LIN {X 0,Y 287.469,Z 770.66,A -85,B 0,C 180,E1 15282.197,E2 15282.197} C_VEL
LIN {X 0,Y 284.222,Z 794.755,A -85,B 0,C 180,E1 15292.332,E2 15292.332} C_VEL
LIN {X 0,Y 283.558,Z 803.475,A -85,B 0,C 180,E1 15301.536,E2 15301.536} C_VEL
LIN {X 0,Y 286.517,Z 800.266,A -85,B 0,C 180,E1 15312.078,E2 15312.078} C_VEL
LIN {X 0,Y 295.291,Z 782.461,A -85,B 0,C 180,E1 15322.672,E2 15322.672} C_VEL
LIN {X 0,Y 310.882,Z 750.712,A -85,B 0,C 180,E1 15331.653,E2 15331.653} C_VEL
LIN {X 0,Y 330.925,Z 705.593,A -85,B 0,C 180,E1 15338.602,E2 15338.602} C_VEL
LIN {X 0,Y 336.814,Z 689.201,A -85,B 0,C 180,E1 15340.792,E2 15340.792} C_VEL
LIN {X 0,Y 337.476,Z 683.839,A -85,B 0,C 180,E1 15344.187,E2 15344.187} C_VEL
LIN {X 0,Y 338.249,Z 688.288,A -85,B 0,C 180,E1 15347.754,E2 15347.754} C_VEL
LIN {X 0,Y 313.848,Z 750.158,A -85,B 0,C 180,E1 15354.353,E2 15354.353} C_VEL
LIN {X 0,Y 295.88,Z 793.344,A -85,B 0,C 180,E1 15362.953,E2 15362.953} C_VEL
LIN {X 0,Y 286.115,Z 820.837,A -85,B 0,C 180,E1 15373.067,E2 15373.067} C_VEL
LIN {X 0,Y 283.836,Z 832.792,A -85,B 0,C 180,E1 15382.345,E2 15382.345} C_VEL
LIN {X 0,Y 283.962,Z 833.571,A -85,B 0,C 180,E1 15391.556,E2 15391.556} C_VEL
LIN {X 0,Y 284.286,Z 822.206,A -85,B 0,C 180,E1 15400.792,E2 15400.792} C_VEL
LIN {X 0,Y 287.24,Z 796.191,A -85,B 0,C 180,E1 15410.108,E2 15410.108} C_VEL
LIN {X 0,Y 300.181,Z 753.134,A -85,B 0,C 180,E1 15421.206,E2 15421.206} C_VEL
LIN {X 0,Y 316.341,Z 705.619,A -85,B 0,C 180,E1 15427.781,E2 15427.781} C_VEL
LIN {X 0,Y 323.777,Z 675.076,A -85,B 0,C 180,E1 15430.595,E2 15430.595} C_VEL
LIN {X 0,Y 318.954,Z 657.733,A -85,B 0,C 180,E1 15435.308,E2 15435.308} C_VEL
LIN {X 0,Y 315.945,Z 652.697,A -85,B 0,C 180,E1 15439.832,E2 15439.832} C_VEL
LIN {X 0,Y 312.951,Z 664.798,A -85,B 0,C 180,E1 15445.963,E2 15445.963} C_VEL
LIN {X 0,Y 312.289,Z 682.68,A -85,B 0,C 180,E1 15451.384,E2 15451.384} C_VEL
LIN {X 0,Y 297.451,Z 717.791,A -85,B 0,C 180,E1 15458.29,E2 15458.29} C_VEL
LIN {X 0,Y 286.13,Z 736.914,A -85,B 0,C 180,E1 15466.19,E2 15466.19} C_VEL
LIN {X 0,Y 279.764,Z 741.327,A -85,B 0,C 180,E1 15475.331,E2 15475.331} C_VEL
LIN {X 0,Y 278.19,Z 731.042,A -85,B 0,C 180,E1 15483.907,E2 15483.907} C_VEL
LIN {X 0,Y 279.775,Z 705.474,A -85,B 0,C 180,E1 15492.228,E2 15492.228} C_VEL
LIN {X 0,Y 283.473,Z 665.617,A -85,B 0,C 180,E1 15498.935,E2 15498.935} C_VEL
LIN {X 0,Y 281.601,Z 639.243,A -85,B 0,C 180,E1 15501.747,E2 15501.747} C_VEL
LIN {X 0,Y 273.533,Z 602.81,A -85,B 0,C 180,E1 15504.584,E2 15504.584} C_VEL
LIN {X 0,Y 272.564,Z 602.81,A -85,B 0,C 180,E1 15516.131,E2 15516.131} C_VEL
LIN {X 0,Y 272.447,Z 602.81,A -85,B 0,C 180,E1 15530.139,E2 15530.139} C_VEL
LIN {X 0,Y 272.833,Z 602.81,A -85,B 0,C 180,E1 15541.759,E2 15541.759} C_VEL
LIN {X 0,Y 273.836,Z 602.81,A -85,B 0,C 180,E1 15555.866,E2 15555.866} C_VEL
LIN {X 0,Y 275.222,Z 602.81,A -85,B 0,C 180,E1 15568.395,E2 15568.395} C_VEL
LIN {X 0,Y 274.237,Z 602.81,A -85,B 0,C 180,E1 15581.14,E2 15581.14} C_VEL
LIN {X 0,Y 273.286,Z 602.81,A -85,B 0,C 180,E1 15594.58,E2 15594.58} C_VEL
LIN {X 0,Y 272.71,Z 602.81,A -85,B 0,C 180,E1 15606.216,E2 15606.216} C_VEL
LIN {X 0,Y 272.978,Z 604.085,A -85,B 0,C 180,E1 15619.483,E2 15619.483} C_VEL
LIN {X 0,Y 292.995,Z 665.219,A -85,B 0,C 180,E1 15624.943,E2 15624.943} C_VEL
LIN {X 0,Y 295.039,Z 684.173,A -85,B 0,C 180,E1 15626.919,E2 15626.919} C_VEL
LIN {X 0,Y 286.379,Z 734.413,A -85,B 0,C 180,E1 15633.535,E2 15633.535} C_VEL
LIN {X 0,Y 279.424,Z 771.619,A -85,B 0,C 180,E1 15642.226,E2 15642.226} C_VEL
LIN {X 0,Y 276.273,Z 794.637,A -85,B 0,C 180,E1 15652.11,E2 15652.11} C_VEL
LIN {X 0,Y 275.575,Z 803.87,A -85,B 0,C 180,E1 15661.58,E2 15661.58} C_VEL
LIN {X 0,Y 278.805,Z 801.152,A -85,B 0,C 180,E1 15672.577,E2 15672.577} C_VEL
LIN {X 0,Y 288.146,Z 784.349,A -85,B 0,C 180,E1 15683.267,E2 15683.267} C_VEL
LIN {X 0,Y 305.45,Z 752.594,A -85,B 0,C 180,E1 15692.705,E2 15692.705} C_VEL
LIN {X 0,Y 327.249,Z 708.48,A -85,B 0,C 180,E1 15699.733,E2 15699.733} C_VEL
LIN {X 0,Y 332.934,Z 695.38,A -85,B 0,C 180,E1 15701.371,E2 15701.371} C_VEL
LIN {X 0,Y 334.073,Z 691.222,A -85,B 0,C 180,E1 15704.757,E2 15704.757} C_VEL
LIN {X 0,Y 334.163,Z 694.797,A -85,B 0,C 180,E1 15707.115,E2 15707.115} C_VEL
LIN {X 0,Y 309.62,Z 749.376,A -85,B 0,C 180,E1 15712.915,E2 15712.915} C_VEL
LIN {X 0,Y 289.453,Z 793.221,A -85,B 0,C 180,E1 15721.877,E2 15721.877} C_VEL
LIN {X 0,Y 278.386,Z 821.027,A -85,B 0,C 180,E1 15732.582,E2 15732.582} C_VEL
LIN {X 0,Y 275.855,Z 832.48,A -85,B 0,C 180,E1 15742.122,E2 15742.122} C_VEL
LIN {X 0,Y 275.993,Z 832.853,A -85,B 0,C 180,E1 15751.601,E2 15751.601} C_VEL
LIN {X 0,Y 276.307,Z 820.985,A -85,B 0,C 180,E1 15761.108,E2 15761.108} C_VEL
LIN {X 0,Y 279.561,Z 794.339,A -85,B 0,C 180,E1 15770.686,E2 15770.686} C_VEL
LIN {X 0,Y 292.103,Z 757.137,A -85,B 0,C 180,E1 15781.346,E2 15781.346} C_VEL
LIN {X 0,Y 309.645,Z 710.546,A -85,B 0,C 180,E1 15788.433,E2 15788.433} C_VEL
LIN {X 0,Y 318.887,Z 677.805,A -85,B 0,C 180,E1 15791.672,E2 15791.672} C_VEL
LIN {X 0,Y 314.799,Z 662.667,A -85,B 0,C 180,E1 15796.655,E2 15796.655} C_VEL
LIN {X 0,Y 312.531,Z 660.915,A -85,B 0,C 180,E1 15803.272,E2 15803.272} C_VEL
LIN {X 0,Y 312.951,Z 664.798,A -85,B 0,C 180,E1 15805.963,E2 15805.963} C_VEL
LIN {X 0,Y 308.353,Z 681.058,A -85,B 0,C 180,E1 15809.107,E2 15809.107} C_VEL
LIN {X 0,Y 300.727,Z 701.492,A -85,B 0,C 180,E1 15812.988,E2 15812.988} C_VEL
LIN {X 0,Y 285.864,Z 729.53,A -85,B 0,C 180,E1 15820.621,E2 15820.621} C_VEL
LIN {X 0,Y 275.928,Z 742.078,A -85,B 0,C 180,E1 15828.9,E2 15828.9} C_VEL
LIN {X 0,Y 271.169,Z 740.21,A -85,B 0,C 180,E1 15838.394,E2 15838.394} C_VEL
LIN {X 0,Y 270.306,Z 723.721,A -85,B 0,C 180,E1 15847.254,E2 15847.254} C_VEL
LIN {X 0,Y 272.947,Z 691.929,A -85,B 0,C 180,E1 15855.31,E2 15855.31} C_VEL
LIN {X 0,Y 275.844,Z 650.722,A -85,B 0,C 180,E1 15860.949,E2 15860.949} C_VEL
LIN {X 0,Y 265.38,Z 602.81,A -85,B 0,C 180,E1 15865.13,E2 15865.13} C_VEL
LIN {X 0,Y 264.414,Z 602.81,A -85,B 0,C 180,E1 15879.179,E2 15879.179} C_VEL
LIN {X 0,Y 264.42,Z 602.81,A -85,B 0,C 180,E1 15892.915,E2 15892.915} C_VEL
LIN {X 0,Y 264.872,Z 602.81,A -85,B 0,C 180,E1 15904.525,E2 15904.525} C_VEL
LIN {X 0,Y 266.041,Z 602.81,A -85,B 0,C 180,E1 15918.458,E2 15918.458} C_VEL
LIN {X 0,Y 266.94,Z 602.81,A -85,B 0,C 180,E1 15931.602,E2 15931.602} C_VEL
LIN {X 0,Y 265.894,Z 602.81,A -85,B 0,C 180,E1 15944.853,E2 15944.853} C_VEL
LIN {X 0,Y 265.023,Z 602.81,A -85,B 0,C 180,E1 15957.445,E2 15957.445} C_VEL
LIN {X 0,Y 264.599,Z 602.81,A -85,B 0,C 180,E1 15971.224,E2 15971.224} C_VEL
LIN {X 0,Y 264.888,Z 603.872,A -85,B 0,C 180,E1 15978.645,E2 15978.645} C_VEL
LIN {X 0,Y 284.837,Z 664.739,A -85,B 0,C 180,E1 15984.251,E2 15984.251} C_VEL
LIN {X 0,Y 287.376,Z 685.203,A -85,B 0,C 180,E1 15986.469,E2 15986.469} C_VEL
LIN {X 0,Y 278.443,Z 735.564,A -85,B 0,C 180,E1 15993.321,E2 15993.321} C_VEL
LIN {X 0,Y 271.266,Z 773.261,A -85,B 0,C 180,E1 16002.504,E2 16002.504} C_VEL
LIN {X 0,Y 268.205,Z 795.774,A -85,B 0,C 180,E1 16012.689,E2 16012.689} C_VEL
LIN {X 0,Y 267.587,Z 804.24,A -85,B 0,C 180,E1 16021.627,E2 16021.627} C_VEL
LIN {X 0,Y 271.036,Z 802.205,A -85,B 0,C 180,E1 16032.944,E2 16032.944} C_VEL
LIN {X 0,Y 282.031,Z 784.649,A -85,B 0,C 180,E1 16044.647,E2 16044.647} C_VEL
LIN {X 0,Y 301.744,Z 752.031,A -85,B 0,C 180,E1 16054.371,E2 16054.371} C_VEL
LIN {X 0,Y 326.723,Z 706.2,A -85,B 0,C 180,E1 16061.502,E2 16061.502} C_VEL
LIN {X 0,Y 329.631,Z 699.986,A -85,B 0,C 180,E1 16062.496,E2 16062.496} C_VEL
LIN {X 0,Y 330.683,Z 699.253,A -85,B 0,C 180,E1 16066.028,E2 16066.028} C_VEL
LIN {X 0,Y 304.263,Z 751.972,A -85,B 0,C 180,E1 16071.922,E2 16071.922} C_VEL
LIN {X 0,Y 282.512,Z 794.499,A -85,B 0,C 180,E1 16081.122,E2 16081.122} C_VEL
LIN {X 0,Y 270.691,Z 821.198,A -85,B 0,C 180,E1 16092.071,E2 16092.071} C_VEL
LIN {X 0,Y 267.82,Z 832.451,A -85,B 0,C 180,E1 16102.568,E2 16102.568} C_VEL
LIN {X 0,Y 268.044,Z 832.084,A -85,B 0,C 180,E1 16111.648,E2 16111.648} C_VEL
LIN {X 0,Y 268.378,Z 819.679,A -85,B 0,C 180,E1 16121.44,E2 16121.44} C_VEL
LIN {X 0,Y 281.539,Z 767.173,A -85,B 0,C 180,E1 16139.932,E2 16139.932} C_VEL
LIN {X 0,Y 298.719,Z 725.735,A -85,B 0,C 180,E1 16147.805,E2 16147.805} C_VEL
LIN {X 0,Y 314.035,Z 681.623,A -85,B 0,C 180,E1 16152.674,E2 16152.674} C_VEL
LIN {X 0,Y 310.873,Z 668.739,A -85,B 0,C 180,E1 16157.638,E2 16157.638} C_VEL
LIN {X 0,Y 309.011,Z 669.222,A -85,B 0,C 180,E1 16164.156,E2 16164.156} C_VEL
LIN {X 0,Y 308.353,Z 681.058,A -85,B 0,C 180,E1 16169.107,E2 16169.107} C_VEL
LIN {X 0,Y 297.981,Z 699.899,A -85,B 0,C 180,E1 16171.12,E2 16171.12} C_VEL
LIN {X 0,Y 281.339,Z 728.984,A -85,B 0,C 180,E1 16178.647,E2 16178.647} C_VEL
LIN {X 0,Y 269.649,Z 742.928,A -85,B 0,C 180,E1 16186.988,E2 16186.988} C_VEL
LIN {X 0,Y 263.562,Z 742.734,A -85,B 0,C 180,E1 16196.697,E2 16196.697} C_VEL
LIN {X 0,Y 262.364,Z 727.153,A -85,B 0,C 180,E1 16206.223,E2 16206.223} C_VEL
LIN {X 0,Y 264.607,Z 696.697,A -85,B 0,C 180,E1 16214.649,E2 16214.649} C_VEL
LIN {X 0,Y 268.302,Z 653.679,A -85,B 0,C 180,E1 16220.996,E2 16220.996} C_VEL
LIN {X 0,Y 257.235,Z 602.81,A -85,B 0,C 180,E1 16225.746,E2 16225.746} C_VEL
LIN {X 0,Y 256.407,Z 602.81,A -85,B 0,C 180,E1 16238.416,E2 16238.416} C_VEL
LIN {X 0,Y 256.424,Z 602.81,A -85,B 0,C 180,E1 16253.022,E2 16253.022} C_VEL
LIN {X 0,Y 256.979,Z 602.81,A -85,B 0,C 180,E1 16267.401,E2 16267.401} C_VEL
LIN {X 0,Y 258.297,Z 602.81,A -85,B 0,C 180,E1 16281.527,E2 16281.527} C_VEL
LIN {X 0,Y 258.955,Z 602.81,A -85,B 0,C 180,E1 16291.651,E2 16291.651} C_VEL
LIN {X 0,Y 257.807,Z 602.81,A -85,B 0,C 180,E1 16305.33,E2 16305.33} C_VEL
LIN {X 0,Y 257.047,Z 602.81,A -85,B 0,C 180,E1 16316.247,E2 16316.247} C_VEL
LIN {X 0,Y 256.544,Z 602.81,A -85,B 0,C 180,E1 16328.356,E2 16328.356} C_VEL
LIN {X 0,Y 256.908,Z 604.687,A -85,B 0,C 180,E1 16337.833,E2 16337.833} C_VEL
LIN {X 0,Y 276.651,Z 664.319,A -85,B 0,C 180,E1 16343.539,E2 16343.539} C_VEL
LIN {X 0,Y 279.656,Z 686.55,A -85,B 0,C 180,E1 16346.047,E2 16346.047} C_VEL
LIN {X 0,Y 270.659,Z 735.793,A -85,B 0,C 180,E1 16352.94,E2 16352.94} C_VEL
LIN {X 0,Y 263.268,Z 773.811,A -85,B 0,C 180,E1 16362.454,E2 16362.454} C_VEL
LIN {X 0,Y 260.096,Z 796.908,A -85,B 0,C 180,E1 16373.361,E2 16373.361} C_VEL
LIN {X 0,Y 259.598,Z 804.598,A -85,B 0,C 180,E1 16381.677,E2 16381.677} C_VEL
LIN {X 0,Y 263.289,Z 803.29,A -85,B 0,C 180,E1 16393.332,E2 16393.332} C_VEL
LIN {X 0,Y 275.056,Z 786.755,A -85,B 0,C 180,E1 16405.316,E2 16405.316} C_VEL
LIN {X 0,Y 296.941,Z 754.215,A -85,B 0,C 180,E1 16415.545,E2 16415.545} C_VEL
LIN {X 0,Y 324.272,Z 709.128,A -85,B 0,C 180,E1 16422.733,E2 16422.733} C_VEL
LIN {X 0,Y 326.195,Z 705.607,A -85,B 0,C 180,E1 16423.893,E2 16423.893} C_VEL
LIN {X 0,Y 325.813,Z 706.997,A -85,B 0,C 180,E1 16425.196,E2 16425.196} C_VEL
LIN {X 0,Y 298.501,Z 755.637,A -85,B 0,C 180,E1 16431.05,E2 16431.05} C_VEL
LIN {X 0,Y 274.994,Z 797.097,A -85,B 0,C 180,E1 16440.708,E2 16440.708} C_VEL
LIN {X 0,Y 262.288,Z 823.151,A -85,B 0,C 180,E1 16452.68,E2 16452.68} C_VEL
LIN {X 0,Y 259.893,Z 831.729,A -85,B 0,C 180,E1 16461.635,E2 16461.635} C_VEL
LIN {X 0,Y 260.078,Z 831.237,A -85,B 0,C 180,E1 16471.699,E2 16471.699} C_VEL
LIN {X 0,Y 260.423,Z 818.323,A -85,B 0,C 180,E1 16481.795,E2 16481.795} C_VEL
LIN {X 0,Y 275.82,Z 764.726,A -85,B 0,C 180,E1 16501.538,E2 16501.538} C_VEL
LIN {X 0,Y 295.082,Z 722.453,A -85,B 0,C 180,E1 16509.512,E2 16509.512} C_VEL
LIN {X 0,Y 309.243,Z 685.758,A -85,B 0,C 180,E1 16513.651,E2 16513.651} C_VEL
LIN {X 0,Y 307.017,Z 675.555,A -85,B 0,C 180,E1 16518.141,E2 16518.141} C_VEL
LIN {X 0,Y 304.98,Z 677.854,A -85,B 0,C 180,E1 16525.094,E2 16525.094} C_VEL
LIN {X 0,Y 301.801,Z 692.035,A -85,B 0,C 180,E1 16529.805,E2 16529.805} C_VEL
LIN {X 0,Y 297.981,Z 699.899,A -85,B 0,C 180,E1 16531.12,E2 16531.12} C_VEL
LIN {X 0,Y 284.761,Z 717.187,A -85,B 0,C 180,E1 16533.109,E2 16533.109} C_VEL
LIN {X 0,Y 268.1,Z 739.787,A -85,B 0,C 180,E1 16541.859,E2 16541.859} C_VEL
LIN {X 0,Y 258.235,Z 746.307,A -85,B 0,C 180,E1 16551.55,E2 16551.55} C_VEL
LIN {X 0,Y 254.341,Z 738.641,A -85,B 0,C 180,E1 16560.852,E2 16560.852} C_VEL
LIN {X 0,Y 254.813,Z 716.975,A -85,B 0,C 180,E1 16569.941,E2 16569.941} C_VEL
LIN {X 0,Y 258.316,Z 681.012,A -85,B 0,C 180,E1 16577.74,E2 16577.74} C_VEL
LIN {X 0,Y 259.305,Z 648.919,A -85,B 0,C 180,E1 16581.909,E2 16581.909} C_VEL
LIN {X 0,Y 249.167,Z 602.81,A -85,B 0,C 180,E1 16586.093,E2 16586.093} C_VEL
LIN {X 0,Y 248.259,Z 602.81,A -85,B 0,C 180,E1 16600.138,E2 16600.138} C_VEL
LIN {X 0,Y 248.454,Z 602.81,A -85,B 0,C 180,E1 16615.536,E2 16615.536} C_VEL
LIN {X 0,Y 249.223,Z 602.81,A -85,B 0,C 180,E1 16630.686,E2 16630.686} C_VEL
LIN {X 0,Y 250.622,Z 602.81,A -85,B 0,C 180,E1 16644.761,E2 16644.761} C_VEL
LIN {X 0,Y 250.703,Z 602.81,A -85,B 0,C 180,E1 16655.18,E2 16655.18} C_VEL
LIN {X 0,Y 249.457,Z 602.81,A -85,B 0,C 180,E1 16669.515,E2 16669.515} C_VEL
LIN {X 0,Y 248.59,Z 602.81,A -85,B 0,C 180,E1 16684.509,E2 16684.509} C_VEL
LIN {X 0,Y 248.68,Z 604.118,A -85,B 0,C 180,E1 16696.888,E2 16696.888} C_VEL
LIN {X 0,Y 268.789,Z 665.113,A -85,B 0,C 180,E1 16702.941,E2 16702.941} C_VEL
LIN {X 0,Y 271.898,Z 688.181,A -85,B 0,C 180,E1 16705.647,E2 16705.647} C_VEL
LIN {X 0,Y 262.515,Z 737.945,A -85,B 0,C 180,E1 16712.926,E2 16712.926} C_VEL
LIN {X 0,Y 255.286,Z 774.347,A -85,B 0,C 180,E1 16722.417,E2 16722.417} C_VEL
LIN {X 0,Y 252.05,Z 797.428,A -85,B 0,C 180,E1 16733.644,E2 16733.644} C_VEL
LIN {X 0,Y 252.274,Z 806.144,A -85,B 0,C 180,E1 16745.179,E2 16745.179} C_VEL
LIN {X 0,Y 257.768,Z 801.717,A -85,B 0,C 180,E1 16757.121,E2 16757.121} C_VEL
LIN {X 0,Y 273.27,Z 782.144,A -85,B 0,C 180,E1 16769.074,E2 16769.074} C_VEL
LIN {X 0,Y 300.349,Z 745.184,A -85,B 0,C 180,E1 16779.167,E2 16779.167} C_VEL
LIN {X 0,Y 321.944,Z 712.844,A -85,B 0,C 180,E1 16784.193,E2 16784.193} C_VEL
LIN {X 0,Y 291.755,Z 761.023,A -85,B 0,C 180,E1 16790.456,E2 16790.456} C_VEL
LIN {X 0,Y 266.81,Z 800.691,A -85,B 0,C 180,E1 16800.657,E2 16800.657} C_VEL
LIN {X 0,Y 253.97,Z 824.758,A -85,B 0,C 180,E1 16813.267,E2 16813.267} C_VEL
LIN {X 0,Y 251.82,Z 832.288,A -85,B 0,C 180,E1 16824.843,E2 16824.843} C_VEL
LIN {X 0,Y 252.078,Z 827.384,A -85,B 0,C 180,E1 16835.209,E2 16835.209} C_VEL
LIN {X 0,Y 253.512,Z 808.014,A -85,B 0,C 180,E1 16846.165,E2 16846.165} C_VEL
LIN {X 0,Y 269.716,Z 763.882,A -85,B 0,C 180,E1 16862.816,E2 16862.816} C_VEL
LIN {X 0,Y 290.947,Z 721.586,A -85,B 0,C 180,E1 16870.964,E2 16870.964} C_VEL
LIN {X 0,Y 304.515,Z 690.471,A -85,B 0,C 180,E1 16874.523,E2 16874.523} C_VEL
LIN {X 0,Y 303.557,Z 683.416,A -85,B 0,C 180,E1 16877.553,E2 16877.553} C_VEL
LIN {X 0,Y 301.242,Z 682.497,A -85,B 0,C 180,E1 16882.997,E2 16882.997} C_VEL
LIN {X 0,Y 298.273,Z 693.389,A -85,B 0,C 180,E1 16888.242,E2 16888.242} C_VEL
LIN {X 0,Y 284.761,Z 717.187,A -85,B 0,C 180,E1 16893.109,E2 16893.109} C_VEL
LIN {X 0,Y 266.731,Z 736.601,A -85,B 0,C 180,E1 16897.983,E2 16897.983} C_VEL
LIN {X 0,Y 256.462,Z 745.944,A -85,B 0,C 180,E1 16904.555,E2 16904.555} C_VEL
LIN {X 0,Y 248.297,Z 746.231,A -85,B 0,C 180,E1 16914.737,E2 16914.737} C_VEL
LIN {X 0,Y 246.346,Z 732.566,A -85,B 0,C 180,E1 16924.413,E2 16924.413} C_VEL
LIN {X 0,Y 248.209,Z 703.423,A -85,B 0,C 180,E1 16933.701,E2 16933.701} C_VEL
LIN {X 0,Y 252.493,Z 661.404,A -85,B 0,C 180,E1 16940.801,E2 16940.801} C_VEL
LIN {X 0,Y 243.644,Z 613.537,A -85,B 0,C 180,E1 16945.595,E2 16945.595} C_VEL
LIN {X 0,Y 241.048,Z 602.81,A -85,B 0,C 180,E1 16946.573,E2 16946.573} C_VEL
LIN {X 0,Y 240.089,Z 602.81,A -85,B 0,C 180,E1 16961.575,E2 16961.575} C_VEL
LIN {X 0,Y 240.183,Z 602.81,A -85,B 0,C 180,E1 16973.081,E2 16973.081} C_VEL
LIN {X 0,Y 240.787,Z 602.81,A -85,B 0,C 180,E1 16986.031,E2 16986.031} C_VEL
LIN {X 0,Y 242.16,Z 602.81,A -85,B 0,C 180,E1 17000.958,E2 17000.958} C_VEL
LIN {X 0,Y 242.937,Z 602.81,A -85,B 0,C 180,E1 17011.76,E2 17011.76} C_VEL
LIN {X 0,Y 241.631,Z 602.81,A -85,B 0,C 180,E1 17026.384,E2 17026.384} C_VEL
LIN {X 0,Y 240.784,Z 602.81,A -85,B 0,C 180,E1 17038.172,E2 17038.172} C_VEL
LIN {X 0,Y 240.237,Z 602.81,A -85,B 0,C 180,E1 17053.418,E2 17053.418} C_VEL
LIN {X 0,Y 240.72,Z 604.827,A -85,B 0,C 180,E1 17056.002,E2 17056.002} C_VEL
LIN {X 0,Y 260.566,Z 664.509,A -85,B 0,C 180,E1 17062.167,E2 17062.167} C_VEL
LIN {X 0,Y 264.27,Z 688.82,A -85,B 0,C 180,E1 17065.129,E2 17065.129} C_VEL
LIN {X 0,Y 254.74,Z 737.961,A -85,B 0,C 180,E1 17072.509,E2 17072.509} C_VEL
LIN {X 0,Y 247.261,Z 774.98,A -85,B 0,C 180,E1 17082.434,E2 17082.434} C_VEL
LIN {X 0,Y 244.042,Z 797.553,A -85,B 0,C 180,E1 17093.658,E2 17093.658} C_VEL
LIN {X 0,Y 244.333,Z 806.61,A -85,B 0,C 180,E1 17105.348,E2 17105.348} C_VEL
LIN {X 0,Y 250.216,Z 803.048,A -85,B 0,C 180,E1 17117.655,E2 17117.655} C_VEL
LIN {X 0,Y 268.221,Z 782.957,A -85,B 0,C 180,E1 17130.612,E2 17130.612} C_VEL
LIN {X 0,Y 297.394,Z 747.152,A -85,B 0,C 180,E1 17140.588,E2 17140.588} C_VEL
LIN {X 0,Y 312.371,Z 727.33,A -85,B 0,C 180,E1 17144.012,E2 17144.012} C_VEL
LIN {X 0,Y 280.718,Z 772.226,A -85,B 0,C 180,E1 17151.103,E2 17151.103} C_VEL
LIN {X 0,Y 255.476,Z 808.683,A -85,B 0,C 180,E1 17162.625,E2 17162.625} C_VEL
LIN {X 0,Y 245.022,Z 827.676,A -85,B 0,C 180,E1 17175.688,E2 17175.688} C_VEL
LIN {X 0,Y 244.11,Z 831.27,A -85,B 0,C 180,E1 17188.248,E2 17188.248} C_VEL
LIN {X 0,Y 244.347,Z 821.656,A -85,B 0,C 180,E1 17198.96,E2 17198.96} C_VEL
LIN {X 0,Y 260.544,Z 769.201,A -85,B 0,C 180,E1 17222.375,E2 17222.375} C_VEL
LIN {X 0,Y 282.212,Z 730.197,A -85,B 0,C 180,E1 17231.115,E2 17231.115} C_VEL
LIN {X 0,Y 299.81,Z 693.903,A -85,B 0,C 180,E1 17235.894,E2 17235.894} C_VEL
LIN {X 0,Y 297.859,Z 688.873,A -85,B 0,C 180,E1 17240.441,E2 17240.441} C_VEL
LIN {X 0,Y 295.178,Z 694.354,A -85,B 0,C 180,E1 17246.09,E2 17246.09} C_VEL
LIN {X 0,Y 286.059,Z 710.478,A -85,B 0,C 180,E1 17249.735,E2 17249.735} C_VEL
LIN {X 0,Y 266.731,Z 736.601,A -85,B 0,C 180,E1 17257.983,E2 17257.983} C_VEL
LIN {X 0,Y 248.864,Z 748.149,A -85,B 0,C 180,E1 17264.252,E2 17264.252} C_VEL
LIN {X 0,Y 240.413,Z 747.312,A -85,B 0,C 180,E1 17274.564,E2 17274.564} C_VEL
LIN {X 0,Y 238.376,Z 731.695,A -85,B 0,C 180,E1 17285.019,E2 17285.019} C_VEL
LIN {X 0,Y 240.368,Z 702.456,A -85,B 0,C 180,E1 17294.157,E2 17294.157} C_VEL
LIN {X 0,Y 244.851,Z 659.209,A -85,B 0,C 180,E1 17301.425,E2 17301.425} C_VEL
LIN {X 0,Y 234.357,Z 608.979,A -85,B 0,C 180,E1 17306.393,E2 17306.393} C_VEL
LIN {X 0,Y 232.97,Z 602.81,A -85,B 0,C 180,E1 17307.077,E2 17307.077} C_VEL
LIN {X 0,Y 232.086,Z 602.81,A -85,B 0,C 180,E1 17323.352,E2 17323.352} C_VEL
LIN {X 0,Y 232.202,Z 602.81,A -85,B 0,C 180,E1 17336.222,E2 17336.222} C_VEL
LIN {X 0,Y 233.017,Z 602.81,A -85,B 0,C 180,E1 17350.775,E2 17350.775} C_VEL
LIN {X 0,Y 234.514,Z 602.81,A -85,B 0,C 180,E1 17364.4,E2 17364.4} C_VEL
LIN {X 0,Y 234.617,Z 602.81,A -85,B 0,C 180,E1 17375.537,E2 17375.537} C_VEL
LIN {X 0,Y 233.314,Z 602.81,A -85,B 0,C 180,E1 17389.433,E2 17389.433} C_VEL
LIN {X 0,Y 232.341,Z 602.81,A -85,B 0,C 180,E1 17403.682,E2 17403.682} C_VEL
LIN {X 0,Y 232.529,Z 604.282,A -85,B 0,C 180,E1 17414.985,E2 17414.985} C_VEL
LIN {X 0,Y 252.73,Z 665.265,A -85,B 0,C 180,E1 17421.531,E2 17421.531} C_VEL
LIN {X 0,Y 256.596,Z 689.709,A -85,B 0,C 180,E1 17424.627,E2 17424.627} C_VEL
LIN {X 0,Y 246.761,Z 738.972,A -85,B 0,C 180,E1 17432.289,E2 17432.289} C_VEL
LIN {X 0,Y 239.246,Z 775.446,A -85,B 0,C 180,E1 17442.41,E2 17442.41} C_VEL
LIN {X 0,Y 235.949,Z 798.618,A -85,B 0,C 180,E1 17454.467,E2 17454.467} C_VEL
LIN {X 0,Y 236.521,Z 807.274,A -85,B 0,C 180,E1 17466.356,E2 17466.356} C_VEL
LIN {X 0,Y 244.405,Z 802.877,A -85,B 0,C 180,E1 17479.97,E2 17479.97} C_VEL
LIN {X 0,Y 265.226,Z 782.172,A -85,B 0,C 180,E1 17492.928,E2 17492.928} C_VEL
LIN {X 0,Y 298.534,Z 745.063,A -85,B 0,C 180,E1 17502.836,E2 17502.836} C_VEL
LIN {X 0,Y 301.86,Z 741.197,A -85,B 0,C 180,E1 17503.979,E2 17503.979} C_VEL
LIN {X 0,Y 267.512,Z 784.783,A -85,B 0,C 180,E1 17512.565,E2 17512.565} C_VEL
LIN {X 0,Y 244.85,Z 814.895,A -85,B 0,C 180,E1 17524.652,E2 17524.652} C_VEL
LIN {X 0,Y 236.622,Z 828.828,A -85,B 0,C 180,E1 17537.061,E2 17537.061} C_VEL
LIN {X 0,Y 236.145,Z 830.46,A -85,B 0,C 180,E1 17548.189,E2 17548.189} C_VEL
LIN {X 0,Y 236.441,Z 820.294,A -85,B 0,C 180,E1 17559.263,E2 17559.263} C_VEL
LIN {X 0,Y 240.889,Z 792.817,A -85,B 0,C 180,E1 17573.216,E2 17573.216} C_VEL
LIN {X 0,Y 258.037,Z 762.731,A -85,B 0,C 180,E1 17585.533,E2 17585.533} C_VEL
LIN {X 0,Y 283.287,Z 721.322,A -85,B 0,C 180,E1 17593.9,E2 17593.9} C_VEL
LIN {X 0,Y 295.167,Z 698.541,A -85,B 0,C 180,E1 17596.929,E2 17596.929} C_VEL
LIN {X 0,Y 292.169,Z 696.888,A -85,B 0,C 180,E1 17603.649,E2 17603.649} C_VEL
LIN {X 0,Y 287.696,Z 704.996,A -85,B 0,C 180,E1 17606.82,E2 17606.82} C_VEL
LIN {X 0,Y 265.479,Z 733.909,A -85,B 0,C 180,E1 17614.612,E2 17614.612} C_VEL
LIN {X 0,Y 248.864,Z 748.149,A -85,B 0,C 180,E1 17624.252,E2 17624.252} C_VEL
LIN {X 0,Y 234.089,Z 749.971,A -85,B 0,C 180,E1 17631.849,E2 17631.849} C_VEL
LIN {X 0,Y 230.28,Z 736.729,A -85,B 0,C 180,E1 17642.83,E2 17642.83} C_VEL
LIN {X 0,Y 231.888,Z 709.009,A -85,B 0,C 180,E1 17652.757,E2 17652.757} C_VEL
LIN {X 0,Y 236.237,Z 667.516,A -85,B 0,C 180,E1 17660.686,E2 17660.686} C_VEL
LIN {X 0,Y 231.775,Z 632.588,A -85,B 0,C 180,E1 17664.87,E2 17664.87} C_VEL
LIN {X 0,Y 224.871,Z 602.81,A -85,B 0,C 180,E1 17667.685,E2 17667.685} C_VEL
LIN {X 0,Y 224,Z 602.81,A -85,B 0,C 180,E1 17680.055,E2 17680.055} C_VEL
LIN {X 0,Y 224.127,Z 602.81,A -85,B 0,C 180,E1 17694.83,E2 17694.83} C_VEL
LIN {X 0,Y 224.745,Z 602.81,A -85,B 0,C 180,E1 17708.168,E2 17708.168} C_VEL
LIN {X 0,Y 225.992,Z 602.81,A -85,B 0,C 180,E1 17720.305,E2 17720.305} C_VEL
LIN {X 0,Y 226.919,Z 602.81,A -85,B 0,C 180,E1 17731.885,E2 17731.885} C_VEL
LIN {X 0,Y 225.761,Z 602.81,A -85,B 0,C 180,E1 17743.573,E2 17743.573} C_VEL
LIN {X 0,Y 224.772,Z 602.81,A -85,B 0,C 180,E1 17755.992,E2 17755.992} C_VEL
LIN {X 0,Y 224.135,Z 602.81,A -85,B 0,C 180,E1 17769.985,E2 17769.985} C_VEL
LIN {X 0,Y 224.512,Z 604.63,A -85,B 0,C 180,E1 17773.996,E2 17773.996} C_VEL
LIN {X 0,Y 244.701,Z 665.156,A -85,B 0,C 180,E1 17780.769,E2 17780.769} C_VEL
LIN {X 0,Y 248.908,Z 690.558,A -85,B 0,C 180,E1 17784.113,E2 17784.113} C_VEL
LIN {X 0,Y 238.891,Z 739.338,A -85,B 0,C 180,E1 17791.938,E2 17791.938} C_VEL
LIN {X 0,Y 231.051,Z 776.924,A -85,B 0,C 180,E1 17802.813,E2 17802.813} C_VEL
LIN {X 0,Y 227.891,Z 799.344,A -85,B 0,C 180,E1 17815.075,E2 17815.075} C_VEL
LIN {X 0,Y 228.439,Z 807.495,A -85,B 0,C 180,E1 17825.722,E2 17825.722} C_VEL
LIN {X 0,Y 235.192,Z 805.594,A -85,B 0,C 180,E1 17838.823,E2 17838.823} C_VEL
LIN {X 0,Y 255.397,Z 788.458,A -85,B 0,C 180,E1 17852.33,E2 17852.33} C_VEL
LIN {X 0,Y 289.975,Z 754.552,A -85,B 0,C 180,E1 17862.951,E2 17862.951} C_VEL
LIN {X 0,Y 291.096,Z 753.63,A -85,B 0,C 180,E1 17864.037,E2 17864.037} C_VEL
LIN {X 0,Y 254.906,Z 794.862,A -85,B 0,C 180,E1 17874.032,E2 17874.032} C_VEL
LIN {X 0,Y 234.238,Z 820.241,A -85,B 0,C 180,E1 17887.161,E2 17887.161} C_VEL
LIN {X 0,Y 228.008,Z 830.067,A -85,B 0,C 180,E1 17900.455,E2 17900.455} C_VEL
LIN {X 0,Y 228.27,Z 827.488,A -85,B 0,C 180,E1 17911.936,E2 17911.936} C_VEL
LIN {X 0,Y 228.827,Z 812.117,A -85,B 0,C 180,E1 17923.452,E2 17923.452} C_VEL
LIN {X 0,Y 232.086,Z 795.033,A -85,B 0,C 180,E1 17932.115,E2 17932.115} C_VEL
LIN {X 0,Y 249.087,Z 767.417,A -85,B 0,C 180,E1 17945.395,E2 17945.395} C_VEL
LIN {X 0,Y 275.958,Z 727.639,A -85,B 0,C 180,E1 17954.548,E2 17954.548} C_VEL
LIN {X 0,Y 290.394,Z 704.26,A -85,B 0,C 180,E1 17957.544,E2 17957.544} C_VEL
LIN {X 0,Y 287.197,Z 703.695,A -85,B 0,C 180,E1 17963.698,E2 17963.698} C_VEL
LIN {X 0,Y 282.134,Z 710.989,A -85,B 0,C 180,E1 17966.078,E2 17966.078} C_VEL
LIN {X 0,Y 258.957,Z 737.592,A -85,B 0,C 180,E1 17973.925,E2 17973.925} C_VEL
LIN {X 0,Y 241.491,Z 750.278,A -85,B 0,C 180,E1 17983.731,E2 17983.731} C_VEL
LIN {X 0,Y 234.089,Z 749.971,A -85,B 0,C 180,E1 17991.849,E2 17991.849} C_VEL
LIN {X 0,Y 222.671,Z 741.924,A -85,B 0,C 180,E1 18000.057,E2 18000.057} C_VEL
LIN {X 0,Y 223.034,Z 716.678,A -85,B 0,C 180,E1 18010.781,E2 18010.781} C_VEL
LIN {X 0,Y 227.224,Z 677.627,A -85,B 0,C 180,E1 18019.503,E2 18019.503} C_VEL
LIN {X 0,Y 227.232,Z 650.533,A -85,B 0,C 180,E1 18023.305,E2 18023.305} C_VEL
LIN {X 0,Y 216.757,Z 602.81,A -85,B 0,C 180,E1 18028.197,E2 18028.197} C_VEL
LIN {X 0,Y 215.822,Z 602.81,A -85,B 0,C 180,E1 18042.372,E2 18042.372} C_VEL
LIN {X 0,Y 216.174,Z 602.81,A -85,B 0,C 180,E1 18058.196,E2 18058.196} C_VEL
LIN {X 0,Y 216.997,Z 602.81,A -85,B 0,C 180,E1 18071.625,E2 18071.625} C_VEL
LIN {X 0,Y 218.387,Z 602.81,A -85,B 0,C 180,E1 18083.985,E2 18083.985} C_VEL
LIN {X 0,Y 218.528,Z 602.81,A -85,B 0,C 180,E1 18095.946,E2 18095.946} C_VEL
LIN {X 0,Y 217.101,Z 602.81,A -85,B 0,C 180,E1 18109.342,E2 18109.342} C_VEL
LIN {X 0,Y 216.346,Z 602.81,A -85,B 0,C 180,E1 18121.698,E2 18121.698} C_VEL
LIN {X 0,Y 216.307,Z 604.213,A -85,B 0,C 180,E1 18132.883,E2 18132.883} C_VEL
LIN {X 0,Y 236.688,Z 665.111,A -85,B 0,C 180,E1 18139.986,E2 18139.986} C_VEL
LIN {X 0,Y 241.14,Z 691.817,A -85,B 0,C 180,E1 18143.635,E2 18143.635} C_VEL
LIN {X 0,Y 230.876,Z 740.407,A -85,B 0,C 180,E1 18151.746,E2 18151.746} C_VEL
LIN {X 0,Y 222.858,Z 778.187,A -85,B 0,C 180,E1 18163.182,E2 18163.182} C_VEL
LIN {X 0,Y 219.852,Z 800.397,A -85,B 0,C 180,E1 18176.045,E2 18176.045} C_VEL
LIN {X 0,Y 221.593,Z 808.829,A -85,B 0,C 180,E1 18189.861,E2 18189.861} C_VEL
LIN {X 0,Y 234.237,Z 802.706,A -85,B 0,C 180,E1 18204.907,E2 18204.907} C_VEL
LIN {X 0,Y 258.955,Z 783.054,A -85,B 0,C 180,E1 18216.92,E2 18216.92} C_VEL
LIN {X 0,Y 282.838,Z 761.923,A -85,B 0,C 180,E1 18223.631,E2 18223.631} C_VEL
LIN {X 0,Y 245.921,Z 799.769,A -85,B 0,C 180,E1 18234.151,E2 18234.151} C_VEL
LIN {X 0,Y 225.074,Z 822.649,A -85,B 0,C 180,E1 18248.27,E2 18248.27} C_VEL
LIN {X 0,Y 220.06,Z 829.603,A -85,B 0,C 180,E1 18260.106,E2 18260.106} C_VEL
LIN {X 0,Y 220.289,Z 825.889,A -85,B 0,C 180,E1 18272.694,E2 18272.694} C_VEL
LIN {X 0,Y 221.145,Z 808.82,A -85,B 0,C 180,E1 18284.688,E2 18284.688} C_VEL
LIN {X 0,Y 223.898,Z 795.597,A -85,B 0,C 180,E1 18291.919,E2 18291.919} C_VEL
LIN {X 0,Y 241.596,Z 769.534,A -85,B 0,C 180,E1 18305.986,E2 18305.986} C_VEL
LIN {X 0,Y 269.33,Z 732.57,A -85,B 0,C 180,E1 18315.376,E2 18315.376} C_VEL
LIN {X 0,Y 284.977,Z 709.615,A -85,B 0,C 180,E1 18318.749,E2 18318.749} C_VEL
LIN {X 0,Y 281.247,Z 711.206,A -85,B 0,C 180,E1 18324.069,E2 18324.069} C_VEL
LIN {X 0,Y 254.248,Z 739.629,A -85,B 0,C 180,E1 18332.445,E2 18332.445} C_VEL
LIN {X 0,Y 234.283,Z 752.293,A -85,B 0,C 180,E1 18343.051,E2 18343.051} C_VEL
LIN {X 0,Y 224.661,Z 749.247,A -85,B 0,C 180,E1 18354.182,E2 18354.182} C_VEL
LIN {X 0,Y 222.671,Z 741.924,A -85,B 0,C 180,E1 18360.057,E2 18360.057} C_VEL
LIN {X 0,Y 214.492,Z 725.205,A -85,B 0,C 180,E1 18368.015,E2 18368.015} C_VEL
LIN {X 0,Y 217.739,Z 690.23,A -85,B 0,C 180,E1 18377.487,E2 18377.487} C_VEL
LIN {X 0,Y 219.763,Z 653.813,A -85,B 0,C 180,E1 18383.269,E2 18383.269} C_VEL
LIN {X 0,Y 208.558,Z 602.81,A -85,B 0,C 180,E1 18389.046,E2 18389.046} C_VEL
LIN {X 0,Y 207.648,Z 602.81,A -85,B 0,C 180,E1 18405.989,E2 18405.989} C_VEL
LIN {X 0,Y 208.243,Z 602.81,A -85,B 0,C 180,E1 18421.692,E2 18421.692} C_VEL
LIN {X 0,Y 209.565,Z 602.81,A -85,B 0,C 180,E1 18437.82,E2 18437.82} C_VEL
LIN {X 0,Y 210.881,Z 602.81,A -85,B 0,C 180,E1 18452.028,E2 18452.028} C_VEL
LIN {X 0,Y 209.518,Z 602.81,A -85,B 0,C 180,E1 18464.648,E2 18464.648} C_VEL
LIN {X 0,Y 208.47,Z 602.81,A -85,B 0,C 180,E1 18478.197,E2 18478.197} C_VEL
LIN {X 0,Y 208.363,Z 604.833,A -85,B 0,C 180,E1 18491.818,E2 18491.818} C_VEL
LIN {X 0,Y 228.383,Z 664.17,A -85,B 0,C 180,E1 18499.043,E2 18499.043} C_VEL
LIN {X 0,Y 233.517,Z 692.343,A -85,B 0,C 180,E1 18503.056,E2 18503.056} C_VEL
LIN {X 0,Y 222.894,Z 741.1,A -85,B 0,C 180,E1 18511.478,E2 18511.478} C_VEL
LIN {X 0,Y 214.739,Z 778.781,A -85,B 0,C 180,E1 18523.32,E2 18523.32} C_VEL
LIN {X 0,Y 211.858,Z 800.112,A -85,B 0,C 180,E1 18535.896,E2 18535.896} C_VEL
LIN {X 0,Y 213.714,Z 809.374,A -85,B 0,C 180,E1 18550.228,E2 18550.228} C_VEL
LIN {X 0,Y 227.183,Z 804.468,A -85,B 0,C 180,E1 18565.736,E2 18565.736} C_VEL
LIN {X 0,Y 255.369,Z 784.752,A -85,B 0,C 180,E1 18578.608,E2 18578.608} C_VEL
LIN {X 0,Y 272.577,Z 771.248,A -85,B 0,C 180,E1 18583.176,E2 18583.176} C_VEL
LIN {X 0,Y 230.756,Z 809.8,A -85,B 0,C 180,E1 18597.184,E2 18597.184} C_VEL
LIN {X 0,Y 213.746,Z 827.046,A -85,B 0,C 180,E1 18613.431,E2 18613.431} C_VEL
LIN {X 0,Y 212.261,Z 827.79,A -85,B 0,C 180,E1 18627.985,E2 18627.985} C_VEL
LIN {X 0,Y 212.673,Z 815.708,A -85,B 0,C 180,E1 18640.309,E2 18640.309} C_VEL
LIN {X 0,Y 215.319,Z 796.918,A -85,B 0,C 180,E1 18650.666,E2 18650.666} C_VEL
LIN {X 0,Y 231.881,Z 774.188,A -85,B 0,C 180,E1 18665.482,E2 18665.482} C_VEL
LIN {X 0,Y 261.291,Z 739.008,A -85,B 0,C 180,E1 18675.881,E2 18675.881} C_VEL
LIN {X 0,Y 279.408,Z 715.372,A -85,B 0,C 180,E1 18679.697,E2 18679.697} C_VEL
LIN {X 0,Y 276.905,Z 716.304,A -85,B 0,C 180,E1 18683.125,E2 18683.125} C_VEL
LIN {X 0,Y 249.776,Z 741.798,A -85,B 0,C 180,E1 18690.917,E2 18690.917} C_VEL
LIN {X 0,Y 232.312,Z 752.594,A -85,B 0,C 180,E1 18698.942,E2 18698.942} C_VEL
LIN {X 0,Y 219.374,Z 753.052,A -85,B 0,C 180,E1 18710.038,E2 18710.038} C_VEL
LIN {X 0,Y 214.258,Z 738.771,A -85,B 0,C 180,E1 18722.026,E2 18722.026} C_VEL
LIN {X 0,Y 214.492,Z 725.205,A -85,B 0,C 180,E1 18728.015,E2 18728.015} C_VEL
LIN {X 0,Y 208.648,Z 701.872,A -85,B 0,C 180,E1 18735.11,E2 18735.11} C_VEL
LIN {X 0,Y 212.662,Z 659.107,A -85,B 0,C 180,E1 18742.915,E2 18742.915} C_VEL
LIN {X 0,Y 201.121,Z 605.641,A -85,B 0,C 180,E1 18748.757,E2 18748.757} C_VEL
LIN {X 0,Y 200.47,Z 602.81,A -85,B 0,C 180,E1 18749.47,E2 18749.47} C_VEL
LIN {X 0,Y 199.618,Z 602.81,A -85,B 0,C 180,E1 18766.23,E2 18766.23} C_VEL
LIN {X 0,Y 200.094,Z 602.81,A -85,B 0,C 180,E1 18780.701,E2 18780.701} C_VEL
LIN {X 0,Y 201.189,Z 602.81,A -85,B 0,C 180,E1 18794.658,E2 18794.658} C_VEL
LIN {X 0,Y 202.937,Z 602.81,A -85,B 0,C 180,E1 18807.823,E2 18807.823} C_VEL
LIN {X 0,Y 201.91,Z 602.81,A -85,B 0,C 180,E1 18820.793,E2 18820.793} C_VEL
LIN {X 0,Y 200.62,Z 602.81,A -85,B 0,C 180,E1 18834.542,E2 18834.542} C_VEL
LIN {X 0,Y 200.215,Z 604.824,A -85,B 0,C 180,E1 18850.616,E2 18850.616} C_VEL
LIN {X 0,Y 220.475,Z 664.498,A -85,B 0,C 180,E1 18858.247,E2 18858.247} C_VEL
LIN {X 0,Y 225.66,Z 693.954,A -85,B 0,C 180,E1 18862.596,E2 18862.596} C_VEL
LIN {X 0,Y 214.467,Z 743.707,A -85,B 0,C 180,E1 18871.694,E2 18871.694} C_VEL
LIN {X 0,Y 206.68,Z 778.976,A -85,B 0,C 180,E1 18883.324,E2 18883.324} C_VEL
LIN {X 0,Y 203.857,Z 801.304,A -85,B 0,C 180,E1 18897.176,E2 18897.176} C_VEL
LIN {X 0,Y 205.863,Z 809.82,A -85,B 0,C 180,E1 18910.623,E2 18910.623} C_VEL
LIN {X 0,Y 220.146,Z 806.112,A -85,B 0,C 180,E1 18926.622,E2 18926.622} C_VEL
LIN {X 0,Y 249.71,Z 788.179,A -85,B 0,C 180,E1 18939.652,E2 18939.652} C_VEL
LIN {X 0,Y 262.929,Z 779.038,A -85,B 0,C 180,E1 18943.135,E2 18943.135} C_VEL
LIN {X 0,Y 222.467,Z 812.333,A -85,B 0,C 180,E1 18956.969,E2 18956.969} C_VEL
LIN {X 0,Y 206.994,Z 825.797,A -85,B 0,C 180,E1 18970.775,E2 18970.775} C_VEL
LIN {X 0,Y 203.944,Z 828.197,A -85,B 0,C 180,E1 18983.627,E2 18983.627} C_VEL
LIN {X 0,Y 204.5,Z 820.999,A -85,B 0,C 180,E1 18995.357,E2 18995.357} C_VEL
LIN {X 0,Y 206.588,Z 799.527,A -85,B 0,C 180,E1 19008.274,E2 19008.274} C_VEL
LIN {X 0,Y 222.959,Z 777.245,A -85,B 0,C 180,E1 19025.382,E2 19025.382} C_VEL
LIN {X 0,Y 252.989,Z 745.034,A -85,B 0,C 180,E1 19036.383,E2 19036.383} C_VEL
LIN {X 0,Y 273.163,Z 721.752,A -85,B 0,C 180,E1 19040.491,E2 19040.491} C_VEL
LIN {X 0,Y 270.365,Z 723.508,A -85,B 0,C 180,E1 19042.535,E2 19042.535} C_VEL
LIN {X 0,Y 241.414,Z 746.837,A -85,B 0,C 180,E1 19050.844,E2 19050.844} C_VEL
LIN {X 0,Y 219.542,Z 756.224,A -85,B 0,C 180,E1 19061.875,E2 19061.875} C_VEL
LIN {X 0,Y 208.417,Z 749.647,A -85,B 0,C 180,E1 19074.775,E2 19074.775} C_VEL
LIN {X 0,Y 206.512,Z 728.017,A -85,B 0,C 180,E1 19087.013,E2 19087.013} C_VEL
LIN {X 0,Y 208.648,Z 701.872,A -85,B 0,C 180,E1 19095.11,E2 19095.11} C_VEL
LIN {X 0,Y 204.031,Z 673.879,A -85,B 0,C 180,E1 19101.027,E2 19101.027} C_VEL
LIN {X 0,Y 202.337,Z 647.312,A -85,B 0,C 180,E1 19104.95,E2 19104.95} C_VEL
LIN {X 0,Y 192.373,Z 602.81,A -85,B 0,C 180,E1 19109.737,E2 19109.737} C_VEL
LIN {X 0,Y 191.567,Z 602.81,A -85,B 0,C 180,E1 19127.63,E2 19127.63} C_VEL
LIN {X 0,Y 192.339,Z 602.81,A -85,B 0,C 180,E1 19145.127,E2 19145.127} C_VEL
LIN {X 0,Y 193.633,Z 602.81,A -85,B 0,C 180,E1 19158.665,E2 19158.665} C_VEL
LIN {X 0,Y 194.816,Z 602.81,A -85,B 0,C 180,E1 19172.195,E2 19172.195} C_VEL
LIN {X 0,Y 193.26,Z 602.81,A -85,B 0,C 180,E1 19185.912,E2 19185.912} C_VEL
LIN {X 0,Y 191.993,Z 602.81,A -85,B 0,C 180,E1 19200.868,E2 19200.868} C_VEL
LIN {X 0,Y 192.027,Z 604.399,A -85,B 0,C 180,E1 19209.304,E2 19209.304} C_VEL
LIN {X 0,Y 212.492,Z 664.639,A -85,B 0,C 180,E1 19217.389,E2 19217.389} C_VEL
LIN {X 0,Y 217.815,Z 695.598,A -85,B 0,C 180,E1 19222.141,E2 19222.141} C_VEL
LIN {X 0,Y 206.2,Z 745.372,A -85,B 0,C 180,E1 19231.709,E2 19231.709} C_VEL
LIN {X 0,Y 198.058,Z 781.518,A -85,B 0,C 180,E1 19244.449,E2 19244.449} C_VEL
LIN {X 0,Y 195.881,Z 801.67,A -85,B 0,C 180,E1 19257.784,E2 19257.784} C_VEL
LIN {X 0,Y 197.996,Z 810.258,A -85,B 0,C 180,E1 19271.05,E2 19271.05} C_VEL
LIN {X 0,Y 213.197,Z 807.781,A -85,B 0,C 180,E1 19287.562,E2 19287.562} C_VEL
LIN {X 0,Y 244.144,Z 791.607,A -85,B 0,C 180,E1 19300.744,E2 19300.744} C_VEL
LIN {X 0,Y 252.858,Z 786.301,A -85,B 0,C 180,E1 19303.059,E2 19303.059} C_VEL
LIN {X 0,Y 212.56,Z 815.761,A -85,B 0,C 180,E1 19317.669,E2 19317.669} C_VEL
LIN {X 0,Y 197.301,Z 827.174,A -85,B 0,C 180,E1 19334.422,E2 19334.422} C_VEL
LIN {X 0,Y 196.454,Z 824.395,A -85,B 0,C 180,E1 19350.036,E2 19350.036} C_VEL
LIN {X 0,Y 196.955,Z 810.359,A -85,B 0,C 180,E1 19362.268,E2 19362.268} C_VEL
LIN {X 0,Y 199.11,Z 796.618,A -85,B 0,C 180,E1 19370.093,E2 19370.093} C_VEL
LIN {X 0,Y 216.423,Z 777.527,A -85,B 0,C 180,E1 19386.621,E2 19386.621} C_VEL
LIN {X 0,Y 248.904,Z 746.267,A -85,B 0,C 180,E1 19397.946,E2 19397.946} C_VEL
LIN {X 0,Y 265.109,Z 729.22,A -85,B 0,C 180,E1 19401.64,E2 19401.64} C_VEL
LIN {X 0,Y 235.043,Z 750.352,A -85,B 0,C 180,E1 19409.973,E2 19409.973} C_VEL
LIN {X 0,Y 212.186,Z 758.07,A -85,B 0,C 180,E1 19421.223,E2 19421.223} C_VEL
LIN {X 0,Y 200.92,Z 751.386,A -85,B 0,C 180,E1 19433.492,E2 19433.492} C_VEL
LIN {X 0,Y 198.464,Z 730.409,A -85,B 0,C 180,E1 19446.024,E2 19446.024} C_VEL
LIN {X 0,Y 201.218,Z 695.954,A -85,B 0,C 180,E1 19456.706,E2 19456.706} C_VEL
LIN {X 0,Y 204.031,Z 673.879,A -85,B 0,C 180,E1 19461.027,E2 19461.027} C_VEL
LIN {X 0,Y 193.626,Z 643.904,A -85,B 0,C 180,E1 19465.827,E2 19465.827} C_VEL
LIN {X 0,Y 184.171,Z 602.81,A -85,B 0,C 180,E1 19470.54,E2 19470.54} C_VEL
LIN {X 0,Y 183.367,Z 602.81,A -85,B 0,C 180,E1 19485.247,E2 19485.247} C_VEL
LIN {X 0,Y 183.963,Z 602.81,A -85,B 0,C 180,E1 19502.979,E2 19502.979} C_VEL
LIN {X 0,Y 185.543,Z 602.81,A -85,B 0,C 180,E1 19518.164,E2 19518.164} C_VEL
LIN {X 0,Y 186.786,Z 602.81,A -85,B 0,C 180,E1 19532.29,E2 19532.29} C_VEL
LIN {X 0,Y 185.092,Z 602.81,A -85,B 0,C 180,E1 19546.634,E2 19546.634} C_VEL
LIN {X 0,Y 183.878,Z 602.81,A -85,B 0,C 180,E1 19562.392,E2 19562.392} C_VEL
LIN {X 0,Y 184.01,Z 604.611,A -85,B 0,C 180,E1 19567.986,E2 19567.986} C_VEL
LIN {X 0,Y 204.442,Z 664.58,A -85,B 0,C 180,E1 19576.46,E2 19576.46} C_VEL
LIN {X 0,Y 210.123,Z 696.203,A -85,B 0,C 180,E1 19581.534,E2 19581.534} C_VEL
LIN {X 0,Y 198.193,Z 746.002,A -85,B 0,C 180,E1 19591.479,E2 19591.479} C_VEL
LIN {X 0,Y 190.049,Z 781.296,A -85,B 0,C 180,E1 19604.37,E2 19604.37} C_VEL
LIN {X 0,Y 187.816,Z 802.38,A -85,B 0,C 180,E1 19618.846,E2 19618.846} C_VEL
LIN {X 0,Y 192.672,Z 811.618,A -85,B 0,C 180,E1 19636.005,E2 19636.005} C_VEL
LIN {X 0,Y 212.79,Z 806.963,A -85,B 0,C 180,E1 19652.338,E2 19652.338} C_VEL
LIN {X 0,Y 242.034,Z 793.106,A -85,B 0,C 180,E1 19662.798,E2 19662.798} C_VEL
LIN {X 0,Y 202.765,Z 818.484,A -85,B 0,C 180,E1 19678.451,E2 19678.451} C_VEL
LIN {X 0,Y 189.5,Z 826.726,A -85,B 0,C 180,E1 19693.764,E2 19693.764} C_VEL
LIN {X 0,Y 188.571,Z 823.121,A -85,B 0,C 180,E1 19710.038,E2 19710.038} C_VEL
LIN {X 0,Y 189.185,Z 807.371,A -85,B 0,C 180,E1 19723.37,E2 19723.37} C_VEL
LIN {X 0,Y 191.413,Z 795.382,A -85,B 0,C 180,E1 19730.939,E2 19730.939} C_VEL
LIN {X 0,Y 210.005,Z 777.675,A -85,B 0,C 180,E1 19747.933,E2 19747.933} C_VEL
LIN {X 0,Y 244.408,Z 748.053,A -85,B 0,C 180,E1 19759.418,E2 19759.418} C_VEL
LIN {X 0,Y 254.403,Z 738.661,A -85,B 0,C 180,E1 19761.824,E2 19761.824} C_VEL
LIN {X 0,Y 222.413,Z 756.318,A -85,B 0,C 180,E1 19771.468,E2 19771.468} C_VEL
LIN {X 0,Y 204.812,Z 759.79,A -85,B 0,C 180,E1 19780.521,E2 19780.521} C_VEL
LIN {X 0,Y 192.533,Z 750.573,A -85,B 0,C 180,E1 19794.342,E2 19794.342} C_VEL
LIN {X 0,Y 190.536,Z 726.934,A -85,B 0,C 180,E1 19807.432,E2 19807.432} C_VEL
LIN {X 0,Y 193.928,Z 690.004,A -85,B 0,C 180,E1 19818.236,E2 19818.236} C_VEL
LIN {X 0,Y 196.037,Z 656.952,A -85,B 0,C 180,E1 19824.007,E2 19824.007} C_VEL
LIN {X 0,Y 193.626,Z 643.904,A -85,B 0,C 180,E1 19825.827,E2 19825.827} C_VEL
LIN {X 0,Y 178.818,Z 614.131,A -85,B 0,C 180,E1 19829.704,E2 19829.704} C_VEL
LIN {X 0,Y 176.006,Z 602.81,A -85,B 0,C 180,E1 19831.514,E2 19831.514} C_VEL
LIN {X 0,Y 175.181,Z 602.81,A -85,B 0,C 180,E1 19849.433,E2 19849.433} C_VEL
LIN {X 0,Y 176.184,Z 602.81,A -85,B 0,C 180,E1 19867.154,E2 19867.154} C_VEL
LIN {X 0,Y 177.98,Z 602.81,A -85,B 0,C 180,E1 19882.613,E2 19882.613} C_VEL
LIN {X 0,Y 178.74,Z 602.81,A -85,B 0,C 180,E1 19892.393,E2 19892.393} C_VEL
LIN {X 0,Y 176.984,Z 602.81,A -85,B 0,C 180,E1 19907.42,E2 19907.42} C_VEL
LIN {X 0,Y 175.798,Z 602.81,A -85,B 0,C 180,E1 19926.067,E2 19926.067} C_VEL
LIN {X 0,Y 197.311,Z 667.915,A -85,B 0,C 180,E1 19936.035,E2 19936.035} C_VEL
LIN {X 0,Y 202.147,Z 697.859,A -85,B 0,C 180,E1 19941.065,E2 19941.065} C_VEL
LIN {X 0,Y 190.155,Z 746.598,A -85,B 0,C 180,E1 19951.25,E2 19951.25} C_VEL
LIN {X 0,Y 181.819,Z 782.181,A -85,B 0,C 180,E1 19964.885,E2 19964.885} C_VEL
LIN {X 0,Y 179.797,Z 803.04,A -85,B 0,C 180,E1 19980.004,E2 19980.004} C_VEL
LIN {X 0,Y 184.98,Z 812.151,A -85,B 0,C 180,E1 19996.69,E2 19996.69} C_VEL
LIN {X 0,Y 206.262,Z 808.802,A -85,B 0,C 180,E1 20013.493,E2 20013.493} C_VEL
LIN {X 0,Y 231.558,Z 798.822,A -85,B 0,C 180,E1 20022.693,E2 20022.693} C_VEL
LIN {X 0,Y 193.043,Z 820.59,A -85,B 0,C 180,E1 20039.318,E2 20039.318} C_VEL
LIN {X 0,Y 180.434,Z 826.222,A -85,B 0,C 180,E1 20057.904,E2 20057.904} C_VEL
LIN {X 0,Y 180.814,Z 819.844,A -85,B 0,C 180,E1 20072.444,E2 20072.444} C_VEL
LIN {X 0,Y 181.967,Z 800.698,A -85,B 0,C 180,E1 20086.447,E2 20086.447} C_VEL
LIN {X 0,Y 183.76,Z 794.135,A -85,B 0,C 180,E1 20091.855,E2 20091.855} C_VEL
LIN {X 0,Y 205.609,Z 776.377,A -85,B 0,C 180,E1 20110.266,E2 20110.266} C_VEL
LIN {X 0,Y 243.254,Z 746.974,A -85,B 0,C 180,E1 20122.103,E2 20122.103} C_VEL
LIN {X 0,Y 211.63,Z 760.297,A -85,B 0,C 180,E1 20132.216,E2 20132.216} C_VEL
LIN {X 0,Y 192.246,Z 759.879,A -85,B 0,C 180,E1 20143.959,E2 20143.959} C_VEL
LIN {X 0,Y 183.475,Z 745.977,A -85,B 0,C 180,E1 20157.626,E2 20157.626} C_VEL
LIN {X 0,Y 182.994,Z 717.889,A -85,B 0,C 180,E1 20170.75,E2 20170.75} C_VEL
LIN {X 0,Y 187.869,Z 675.754,A -85,B 0,C 180,E1 20181.31,E2 20181.31} C_VEL
LIN {X 0,Y 186.852,Z 651.144,A -85,B 0,C 180,E1 20185.292,E2 20185.292} C_VEL
LIN {X 0,Y 178.818,Z 614.131,A -85,B 0,C 180,E1 20189.704,E2 20189.704} C_VEL
LIN {X 0,Y 169.8,Z 604,A -85,B 0,C 180,E1 20193.051,E2 20193.051} C_VEL
LIN {X 0,Y 167.312,Z 602.81,A -85,B 0,C 180,E1 20195.542,E2 20195.542} C_VEL
LIN {X 0,Y 167.16,Z 602.81,A -85,B 0,C 180,E1 20213.789,E2 20213.789} C_VEL
LIN {X 0,Y 168.526,Z 602.81,A -85,B 0,C 180,E1 20231.587,E2 20231.587} C_VEL
LIN {X 0,Y 170.707,Z 602.81,A -85,B 0,C 180,E1 20247.411,E2 20247.411} C_VEL
LIN {X 0,Y 169.394,Z 602.81,A -85,B 0,C 180,E1 20262.898,E2 20262.898} C_VEL
LIN {X 0,Y 167.693,Z 602.81,A -85,B 0,C 180,E1 20280.729,E2 20280.729} C_VEL
LIN {X 0,Y 167.978,Z 604.499,A -85,B 0,C 180,E1 20285.031,E2 20285.031} C_VEL
LIN {X 0,Y 188.59,Z 664.922,A -85,B 0,C 180,E1 20294.55,E2 20294.55} C_VEL
LIN {X 0,Y 194.607,Z 697.672,A -85,B 0,C 180,E1 20300.292,E2 20300.292} C_VEL
LIN {X 0,Y 182.25,Z 746.632,A -85,B 0,C 180,E1 20310.87,E2 20310.87} C_VEL
LIN {X 0,Y 173.615,Z 782.987,A -85,B 0,C 180,E1 20325.45,E2 20325.45} C_VEL
LIN {X 0,Y 171.761,Z 803.647,A -85,B 0,C 180,E1 20341.27,E2 20341.27} C_VEL
LIN {X 0,Y 177.318,Z 812.569,A -85,B 0,C 180,E1 20357.433,E2 20357.433} C_VEL
LIN {X 0,Y 203.678,Z 809.543,A -85,B 0,C 180,E1 20376.59,E2 20376.59} C_VEL
LIN {X 0,Y 221.062,Z 803.795,A -85,B 0,C 180,E1 20382.582,E2 20382.582} C_VEL
LIN {X 0,Y 183.207,Z 822.175,A -85,B 0,C 180,E1 20400.431,E2 20400.431} C_VEL
LIN {X 0,Y 172.571,Z 825.311,A -85,B 0,C 180,E1 20417.344,E2 20417.344} C_VEL
LIN {X 0,Y 172.943,Z 818.268,A -85,B 0,C 180,E1 20432.555,E2 20432.555} C_VEL
LIN {X 0,Y 174.563,Z 797.131,A -85,B 0,C 180,E1 20447.755,E2 20447.755} C_VEL
LIN {X 0,Y 199.519,Z 776.495,A -85,B 0,C 180,E1 20471.764,E2 20471.764} C_VEL
LIN {X 0,Y 232.567,Z 753.73,A -85,B 0,C 180,E1 20482.276,E2 20482.276} C_VEL
LIN {X 0,Y 204.898,Z 762.727,A -85,B 0,C 180,E1 20491.22,E2 20491.22} C_VEL
LIN {X 0,Y 184.647,Z 760.894,A -85,B 0,C 180,E1 20503.279,E2 20503.279} C_VEL
LIN {X 0,Y 175.168,Z 744.51,A -85,B 0,C 180,E1 20518.337,E2 20518.337} C_VEL
LIN {X 0,Y 175.321,Z 714.46,A -85,B 0,C 180,E1 20531.859,E2 20531.859} C_VEL
LIN {X 0,Y 180.61,Z 670.896,A -85,B 0,C 180,E1 20542.455,E2 20542.455} C_VEL
LIN {X 0,Y 173.783,Z 627.427,A -85,B 0,C 180,E1 20548.857,E2 20548.857} C_VEL
LIN {X 0,Y 167.899,Z 602.81,A -85,B 0,C 180,E1 20552.02,E2 20552.02} C_VEL
LIN {X 0,Y 167.312,Z 602.81,A -85,B 0,C 180,E1 20555.542,E2 20555.542} C_VEL
LIN {X 0,Y 158.885,Z 602.81,A -85,B 0,C 180,E1 20567.724,E2 20567.724} C_VEL
LIN {X 0,Y 159.763,Z 602.81,A -85,B 0,C 180,E1 20584.649,E2 20584.649} C_VEL
LIN {X 0,Y 161.767,Z 602.81,A -85,B 0,C 180,E1 20601.867,E2 20601.867} C_VEL
LIN {X 0,Y 162.628,Z 602.81,A -85,B 0,C 180,E1 20612.63,E2 20612.63} C_VEL
LIN {X 0,Y 160.637,Z 602.81,A -85,B 0,C 180,E1 20629.259,E2 20629.259} C_VEL
LIN {X 0,Y 159.908,Z 604.465,A -85,B 0,C 180,E1 20643.378,E2 20643.378} C_VEL
LIN {X 0,Y 180.207,Z 663.596,A -85,B 0,C 180,E1 20653.246,E2 20653.246} C_VEL
LIN {X 0,Y 186.558,Z 699.369,A -85,B 0,C 180,E1 20659.794,E2 20659.794} C_VEL
LIN {X 0,Y 173.993,Z 747.824,A -85,B 0,C 180,E1 20670.845,E2 20670.845} C_VEL
LIN {X 0,Y 165.525,Z 783.07,A -85,B 0,C 180,E1 20685.713,E2 20685.713} C_VEL
LIN {X 0,Y 163.813,Z 803.099,A -85,B 0,C 180,E1 20701.331,E2 20701.331} C_VEL
LIN {X 0,Y 169.68,Z 812.926,A -85,B 0,C 180,E1 20718.245,E2 20718.245} C_VEL
LIN {X 0,Y 193.431,Z 812.288,A -85,B 0,C 180,E1 20736.046,E2 20736.046} C_VEL
LIN {X 0,Y 210.353,Z 808.252,A -85,B 0,C 180,E1 20743.162,E2 20743.162} C_VEL
LIN {X 0,Y 176.196,Z 822.174,A -85,B 0,C 180,E1 20759.129,E2 20759.129} C_VEL
LIN {X 0,Y 164.739,Z 824.307,A -85,B 0,C 180,E1 20776.731,E2 20776.731} C_VEL
LIN {X 0,Y 165.086,Z 816.578,A -85,B 0,C 180,E1 20792.677,E2 20792.677} C_VEL
LIN {X 0,Y 166.946,Z 794.434,A -85,B 0,C 180,E1 20808.594,E2 20808.594} C_VEL
LIN {X 0,Y 191.44,Z 777.773,A -85,B 0,C 180,E1 20832.404,E2 20832.404} C_VEL
LIN {X 0,Y 221.472,Z 759.846,A -85,B 0,C 180,E1 20842.041,E2 20842.041} C_VEL
LIN {X 0,Y 189.913,Z 765.338,A -85,B 0,C 180,E1 20853.926,E2 20853.926} C_VEL
LIN {X 0,Y 171.625,Z 756.761,A -85,B 0,C 180,E1 20868.521,E2 20868.521} C_VEL
LIN {X 0,Y 166.425,Z 733.786,A -85,B 0,C 180,E1 20883.917,E2 20883.917} C_VEL
LIN {X 0,Y 169.172,Z 697.323,A -85,B 0,C 180,E1 20896.945,E2 20896.945} C_VEL
LIN {X 0,Y 172.197,Z 659.62,A -85,B 0,C 180,E1 20904.749,E2 20904.749} C_VEL
LIN {X 0,Y 160.36,Z 605.399,A -85,B 0,C 180,E1 20911.854,E2 20911.854} C_VEL
LIN {X 0,Y 159.828,Z 602.81,A -85,B 0,C 180,E1 20912.309,E2 20912.309} C_VEL
LIN {X 0,Y 158.885,Z 602.81,A -85,B 0,C 180,E1 20927.724,E2 20927.724} C_VEL
LIN {X 0,Y 151.257,Z 602.81,A -85,B 0,C 180,E1 20940.623,E2 20940.623} C_VEL
LIN {X 0,Y 152.831,Z 602.81,A -85,B 0,C 180,E1 20955.581,E2 20955.581} C_VEL
LIN {X 0,Y 154.555,Z 602.81,A -85,B 0,C 180,E1 20967.14,E2 20967.14} C_VEL
LIN {X 0,Y 153.838,Z 602.81,A -85,B 0,C 180,E1 20978.462,E2 20978.462} C_VEL
LIN {X 0,Y 151.785,Z 602.81,A -85,B 0,C 180,E1 20996.682,E2 20996.682} C_VEL
LIN {X 0,Y 151.795,Z 603.922,A -85,B 0,C 180,E1 21001.519,E2 21001.519} C_VEL
LIN {X 0,Y 172.508,Z 664.76,A -85,B 0,C 180,E1 21012.316,E2 21012.316} C_VEL
LIN {X 0,Y 178.789,Z 700.004,A -85,B 0,C 180,E1 21019.104,E2 21019.104} C_VEL
LIN {X 0,Y 165.755,Z 748.697,A -85,B 0,C 180,E1 21030.752,E2 21030.752} C_VEL
LIN {X 0,Y 157.272,Z 784.34,A -85,B 0,C 180,E1 21046.757,E2 21046.757} C_VEL
LIN {X 0,Y 155.884,Z 803.591,A -85,B 0,C 180,E1 21062.794,E2 21062.794} C_VEL
LIN {X 0,Y 166.481,Z 814.48,A -85,B 0,C 180,E1 21084.22,E2 21084.22} C_VEL
LIN {X 0,Y 199.915,Z 811.482,A -85,B 0,C 180,E1 21102.387,E2 21102.387} C_VEL
LIN {X 0,Y 166.652,Z 822.723,A -85,B 0,C 180,E1 21119.998,E2 21119.998} C_VEL
LIN {X 0,Y 156.411,Z 821.581,A -85,B 0,C 180,E1 21141.679,E2 21141.679} C_VEL
LIN {X 0,Y 157.258,Z 812.022,A -85,B 0,C 180,E1 21155.582,E2 21155.582} C_VEL
LIN {X 0,Y 159.711,Z 790.655,A -85,B 0,C 180,E1 21170.919,E2 21170.919} C_VEL
LIN {X 0,Y 181.307,Z 779.707,A -85,B 0,C 180,E1 21192.083,E2 21192.083} C_VEL
LIN {X 0,Y 210.168,Z 764.428,A -85,B 0,C 180,E1 21202.773,E2 21202.773} C_VEL
LIN {X 0,Y 182.921,Z 766.996,A -85,B 0,C 180,E1 21212.849,E2 21212.849} C_VEL
LIN {X 0,Y 163.803,Z 756.955,A -85,B 0,C 180,E1 21227.965,E2 21227.965} C_VEL
LIN {X 0,Y 158.493,Z 732.646,A -85,B 0,C 180,E1 21244.114,E2 21244.114} C_VEL
LIN {X 0,Y 161.45,Z 694.503,A -85,B 0,C 180,E1 21257.782,E2 21257.782} C_VEL
LIN {X 0,Y 164.057,Z 659.397,A -85,B 0,C 180,E1 21265.168,E2 21265.168} C_VEL
LIN {X 0,Y 151.59,Z 602.81,A -85,B 0,C 180,E1 21273.401,E2 21273.401} C_VEL
LIN {X 0,Y 150.875,Z 602.81,A -85,B 0,C 180,E1 21289.116,E2 21289.116} C_VEL
LIN {X 0,Y 151.257,Z 602.81,A -85,B 0,C 180,E1 21300.623,E2 21300.623} C_VEL
LIN {X 0,Y 144.53,Z 602.81,A -85,B 0,C 180,E1 21314.245,E2 21314.245} C_VEL
LIN {X 0,Y 146.466,Z 602.81,A -85,B 0,C 180,E1 21326.982,E2 21326.982} C_VEL
LIN {X 0,Y 145.695,Z 602.81,A -85,B 0,C 180,E1 21338.938,E2 21338.938} C_VEL
LIN {X 0,Y 143.628,Z 603.191,A -85,B 0,C 180,E1 21359.445,E2 21359.445} C_VEL
LIN {X 0,Y 164.341,Z 664.043,A -85,B 0,C 180,E1 21370.989,E2 21370.989} C_VEL
LIN {X 0,Y 171.142,Z 700.232,A -85,B 0,C 180,E1 21378.322,E2 21378.322} C_VEL
LIN {X 0,Y 157.501,Z 749.61,A -85,B 0,C 180,E1 21390.711,E2 21390.711} C_VEL
LIN {X 0,Y 149.107,Z 784.88,A -85,B 0,C 180,E1 21407.515,E2 21407.515} C_VEL
LIN {X 0,Y 148.101,Z 804.017,A -85,B 0,C 180,E1 21424.412,E2 21424.412} C_VEL
LIN {X 0,Y 159.208,Z 814.866,A -85,B 0,C 180,E1 21445.403,E2 21445.403} C_VEL
LIN {X 0,Y 190.377,Z 814.099,A -85,B 0,C 180,E1 21462.655,E2 21462.655} C_VEL
LIN {X 0,Y 154.597,Z 823.009,A -85,B 0,C 180,E1 21483.841,E2 21483.841} C_VEL
LIN {X 0,Y 149.068,Z 817.217,A -85,B 0,C 180,E1 21507.13,E2 21507.13} C_VEL
LIN {X 0,Y 149.677,Z 801.799,A -85,B 0,C 180,E1 21522.489,E2 21522.489} C_VEL
LIN {X 0,Y 151.844,Z 788.885,A -85,B 0,C 180,E1 21530.522,E2 21530.522} C_VEL
LIN {X 0,Y 171.21,Z 780.87,A -85,B 0,C 180,E1 21551.714,E2 21551.714} C_VEL
LIN {X 0,Y 199.011,Z 768.249,A -85,B 0,C 180,E1 21562.979,E2 21562.979} C_VEL
LIN {X 0,Y 168.245,Z 766.501,A -85,B 0,C 180,E1 21576.05,E2 21576.05} C_VEL
LIN {X 0,Y 152.801,Z 750.155,A -85,B 0,C 180,E1 21593.008,E2 21593.008} C_VEL
LIN {X 0,Y 150.786,Z 719.901,A -85,B 0,C 180,E1 21609.408,E2 21609.408} C_VEL
LIN {X 0,Y 155.633,Z 677.793,A -85,B 0,C 180,E1 21621.933,E2 21621.933} C_VEL
LIN {X 0,Y 154.958,Z 653.808,A -85,B 0,C 180,E1 21626.535,E2 21626.535} C_VEL
LIN {X 0,Y 143.369,Z 602.81,A -85,B 0,C 180,E1 21634.202,E2 21634.202} C_VEL
LIN {X 0,Y 142.784,Z 602.81,A -85,B 0,C 180,E1 21654.172,E2 21654.172} C_VEL
LIN {X 0,Y 143.826,Z 602.81,A -85,B 0,C 180,E1 21668.278,E2 21668.278} C_VEL
LIN {X 0,Y 144.53,Z 602.81,A -85,B 0,C 180,E1 21674.245,E2 21674.245} C_VEL
LIN {X 0,Y 138.224,Z 602.81,A -85,B 0,C 180,E1 21688.513,E2 21688.513} C_VEL
LIN {X 0,Y 136.618,Z 602.81,A -85,B 0,C 180,E1 21706.067,E2 21706.067} C_VEL
LIN {X 0,Y 135.918,Z 604.799,A -85,B 0,C 180,E1 21717.579,E2 21717.579} C_VEL
LIN {X 0,Y 156.197,Z 663.151,A -85,B 0,C 180,E1 21729.547,E2 21729.547} C_VEL
LIN {X 0,Y 163.305,Z 701.084,A -85,B 0,C 180,E1 21737.618,E2 21737.618} C_VEL
LIN {X 0,Y 149.403,Z 749.852,A -85,B 0,C 180,E1 21750.474,E2 21750.474} C_VEL
LIN {X 0,Y 141.049,Z 785.348,A -85,B 0,C 180,E1 21768.367,E2 21768.367} C_VEL
LIN {X 0,Y 140.771,Z 805.543,A -85,B 0,C 180,E1 21787.749,E2 21787.749} C_VEL
LIN {X 0,Y 158.44,Z 816.349,A -85,B 0,C 180,E1 21811.792,E2 21811.792} C_VEL
LIN {X 0,Y 178.77,Z 816.35,A -85,B 0,C 180,E1 21822.121,E2 21822.121} C_VEL
LIN {X 0,Y 147.41,Z 822.147,A -85,B 0,C 180,E1 21842.46,E2 21842.46} C_VEL
LIN {X 0,Y 141.254,Z 815.452,A -85,B 0,C 180,E1 21866.971,E2 21866.971} C_VEL
LIN {X 0,Y 141.864,Z 800.194,A -85,B 0,C 180,E1 21882.403,E2 21882.403} C_VEL
LIN {X 0,Y 144.341,Z 786.722,A -85,B 0,C 180,E1 21891.641,E2 21891.641} C_VEL
LIN {X 0,Y 169.619,Z 778.391,A -85,B 0,C 180,E1 21915.757,E2 21915.757} C_VEL
LIN {X 0,Y 188.642,Z 771.056,A -85,B 0,C 180,E1 21922.888,E2 21922.888} C_VEL
LIN {X 0,Y 157.563,Z 765.676,A -85,B 0,C 180,E1 21937.337,E2 21937.337} C_VEL
LIN {X 0,Y 143.971,Z 745.589,A -85,B 0,C 180,E1 21955.461,E2 21955.461} C_VEL
LIN {X 0,Y 143.376,Z 712.938,A -85,B 0,C 180,E1 21971.828,E2 21971.828} C_VEL
LIN {X 0,Y 149.067,Z 666.301,A -85,B 0,C 180,E1 21984.574,E2 21984.574} C_VEL
LIN {X 0,Y 137.931,Z 613.479,A -85,B 0,C 180,E1 21993.008,E2 21993.008} C_VEL
LIN {X 0,Y 135.178,Z 602.81,A -85,B 0,C 180,E1 21995.103,E2 21995.103} C_VEL
LIN {X 0,Y 134.549,Z 602.81,A -85,B 0,C 180,E1 22011.598,E2 22011.598} C_VEL
LIN {X 0,Y 136.002,Z 602.81,A -85,B 0,C 180,E1 22031.5,E2 22031.5} C_VEL
LIN {X 0,Y 138.224,Z 602.81,A -85,B 0,C 180,E1 22048.513,E2 22048.513} C_VEL
LIN {X 0,Y 128.659,Z 602.81,A -85,B 0,C 180,E1 22063.396,E2 22063.396} C_VEL
LIN {X 0,Y 128.056,Z 604.877,A -85,B 0,C 180,E1 22075.266,E2 22075.266} C_VEL
LIN {X 0,Y 148.333,Z 663.221,A -85,B 0,C 180,E1 22088.195,E2 22088.195} C_VEL
LIN {X 0,Y 155.475,Z 701.877,A -85,B 0,C 180,E1 22096.869,E2 22096.869} C_VEL
LIN {X 0,Y 141.064,Z 750.778,A -85,B 0,C 180,E1 22110.518,E2 22110.518} C_VEL
LIN {X 0,Y 133.092,Z 784.603,A -85,B 0,C 180,E1 22128.529,E2 22128.529} C_VEL
LIN {X 0,Y 132.902,Z 804.664,A -85,B 0,C 180,E1 22148.211,E2 22148.211} C_VEL
LIN {X 0,Y 151.699,Z 816.739,A -85,B 0,C 180,E1 22173.385,E2 22173.385} C_VEL
LIN {X 0,Y 168.998,Z 817.758,A -85,B 0,C 180,E1 22182.339,E2 22182.339} C_VEL
LIN {X 0,Y 136.198,Z 820.56,A -85,B 0,C 180,E1 22207.106,E2 22207.106} C_VEL
LIN {X 0,Y 133.841,Z 811.291,A -85,B 0,C 180,E1 22230.053,E2 22230.053} C_VEL
LIN {X 0,Y 135.379,Z 789.437,A -85,B 0,C 180,E1 22248.523,E2 22248.523} C_VEL
LIN {X 0,Y 136.955,Z 784.453,A -85,B 0,C 180,E1 22252.872,E2 22252.872} C_VEL
LIN {X 0,Y 164.088,Z 777.461,A -85,B 0,C 180,E1 22277.777,E2 22277.777} C_VEL
LIN {X 0,Y 177.136,Z 773.086,A -85,B 0,C 180,E1 22283.149,E2 22283.149} C_VEL
LIN {X 0,Y 146.951,Z 763.813,A -85,B 0,C 180,E1 22298.807,E2 22298.807} C_VEL
LIN {X 0,Y 135.002,Z 739.567,A -85,B 0,C 180,E1 22318.385,E2 22318.385} C_VEL
LIN {X 0,Y 136.612,Z 702.577,A -85,B 0,C 180,E1 22335.291,E2 22335.291} C_VEL
LIN {X 0,Y 140.171,Z 661.939,A -85,B 0,C 180,E1 22345.791,E2 22345.791} C_VEL
LIN {X 0,Y 127.774,Z 605.891,A -85,B 0,C 180,E1 22354.805,E2 22354.805} C_VEL
LIN {X 0,Y 126.992,Z 602.81,A -85,B 0,C 180,E1 22356.355,E2 22356.355} C_VEL
LIN {X 0,Y 126.703,Z 602.81,A -85,B 0,C 180,E1 22377.324,E2 22377.324} C_VEL
LIN {X 0,Y 129.121,Z 602.81,A -85,B 0,C 180,E1 22399.792,E2 22399.792} C_VEL
LIN {X 0,Y 130.311,Z 602.81,A -85,B 0,C 180,E1 22413.283,E2 22413.283} C_VEL
LIN {X 0,Y 128.659,Z 602.81,A -85,B 0,C 180,E1 22423.396,E2 22423.396} C_VEL
LIN {X 0,Y 119.97,Z 602.81,A -85,B 0,C 180,E1 22429.486,E2 22429.486} C_VEL
LIN {X 0,Y 120.126,Z 605.231,A -85,B 0,C 180,E1 22432.69,E2 22432.69} C_VEL
LIN {X 0,Y 139.456,Z 659.769,A -85,B 0,C 180,E1 22445.912,E2 22445.912} C_VEL
LIN {X 0,Y 147.85,Z 701.912,A -85,B 0,C 180,E1 22455.924,E2 22455.924} C_VEL
LIN {X 0,Y 133.115,Z 750.379,A -85,B 0,C 180,E1 22470.089,E2 22470.089} C_VEL
LIN {X 0,Y 125.017,Z 784.821,A -85,B 0,C 180,E1 22489.515,E2 22489.515} C_VEL
LIN {X 0,Y 125.471,Z 804.868,A -85,B 0,C 180,E1 22510.458,E2 22510.458} C_VEL
LIN {X 0,Y 145.079,Z 817.04,A -85,B 0,C 180,E1 22535.125,E2 22535.125} C_VEL
LIN {X 0,Y 157.674,Z 818.455,A -85,B 0,C 180,E1 22541.853,E2 22541.853} C_VEL
LIN {X 0,Y 128.877,Z 819.23,A -85,B 0,C 180,E1 22565.725,E2 22565.725} C_VEL
LIN {X 0,Y 126.14,Z 809.083,A -85,B 0,C 180,E1 22590.056,E2 22590.056} C_VEL
LIN {X 0,Y 127.997,Z 785.601,A -85,B 0,C 180,E1 22609.986,E2 22609.986} C_VEL
LIN {X 0,Y 129.713,Z 781.947,A -85,B 0,C 180,E1 22614.229,E2 22614.229} C_VEL
LIN {X 0,Y 158.802,Z 776.348,A -85,B 0,C 180,E1 22639.923,E2 22639.923} C_VEL
LIN {X 0,Y 165.477,Z 774.095,A -85,B 0,C 180,E1 22643.406,E2 22643.406} C_VEL
LIN {X 0,Y 136.582,Z 760.987,A -85,B 0,C 180,E1 22660.525,E2 22660.525} C_VEL
LIN {X 0,Y 126.716,Z 733.767,A -85,B 0,C 180,E1 22680.852,E2 22680.852} C_VEL
LIN {X 0,Y 129.379,Z 694.457,A -85,B 0,C 180,E1 22697.812,E2 22697.812} C_VEL
LIN {X 0,Y 131.999,Z 661.509,A -85,B 0,C 180,E1 22706.233,E2 22706.233} C_VEL
LIN {X 0,Y 119.357,Z 604.955,A -85,B 0,C 180,E1 22715.805,E2 22715.805} C_VEL
LIN {X 0,Y 118.541,Z 602.81,A -85,B 0,C 180,E1 22721.097,E2 22721.097} C_VEL
LIN {X 0,Y 118.993,Z 602.81,A -85,B 0,C 180,E1 22743.426,E2 22743.426} C_VEL
LIN {X 0,Y 122.166,Z 602.81,A -85,B 0,C 180,E1 22766.381,E2 22766.381} C_VEL
LIN {X 0,Y 120.598,Z 602.81,A -85,B 0,C 180,E1 22783.086,E2 22783.086} C_VEL
LIN {X 0,Y 119.97,Z 602.81,A -85,B 0,C 180,E1 22789.486,E2 22789.486} C_VEL
LIN {X 0,Y 118.913,Z 612.378,A -85,B 0,C 180,E1 22793.347,E2 22793.347} C_VEL
LIN {X 0,Y 119.781,Z 623.51,A -85,B 0,C 180,E1 22795.293,E2 22795.293} C_VEL
LIN {X 0,Y 135.427,Z 675.022,A -85,B 0,C 180,E1 22807.975,E2 22807.975} C_VEL
LIN {X 0,Y 139.398,Z 704.687,A -85,B 0,C 180,E1 22815.517,E2 22815.517} C_VEL
LIN {X 0,Y 124.342,Z 752.571,A -85,B 0,C 180,E1 22830.786,E2 22830.786} C_VEL
LIN {X 0,Y 116.875,Z 786.115,A -85,B 0,C 180,E1 22851.607,E2 22851.607} C_VEL
LIN {X 0,Y 119.623,Z 807.326,A -85,B 0,C 180,E1 22876.59,E2 22876.59} C_VEL
LIN {X 0,Y 147.591,Z 818.575,A -85,B 0,C 180,E1 22901.943,E2 22901.943} C_VEL
LIN {X 0,Y 118.7,Z 815.787,A -85,B 0,C 180,E1 22931.426,E2 22931.426} C_VEL
LIN {X 0,Y 118.438,Z 805.258,A -85,B 0,C 180,E1 22951.895,E2 22951.895} C_VEL
LIN {X 0,Y 122.058,Z 779.195,A -85,B 0,C 180,E1 22973.893,E2 22973.893} C_VEL
LIN {X 0,Y 152.044,Z 775.342,A -85,B 0,C 180,E1 23001.492,E2 23001.492} C_VEL
LIN {X 0,Y 153.869,Z 774.136,A -85,B 0,C 180,E1 23003.715,E2 23003.715} C_VEL
LIN {X 0,Y 126.283,Z 757.168,A -85,B 0,C 180,E1 23022.512,E2 23022.512} C_VEL
LIN {X 0,Y 118.854,Z 727.058,A -85,B 0,C 180,E1 23043.654,E2 23043.654} C_VEL
LIN {X 0,Y 122.573,Z 684.99,A -85,B 0,C 180,E1 23060.644,E2 23060.644} C_VEL
LIN {X 0,Y 123.718,Z 660.373,A -85,B 0,C 180,E1 23066.812,E2 23066.812} C_VEL
LIN {X 0,Y 110.737,Z 602.81,A -85,B 0,C 180,E1 23078.064,E2 23078.064} C_VEL
LIN {X 0,Y 110.871,Z 602.81,A -85,B 0,C 180,E1 23102.816,E2 23102.816} C_VEL
LIN {X 0,Y 114.048,Z 602.81,A -85,B 0,C 180,E1 23126.21,E2 23126.21} C_VEL
LIN {X 0,Y 112.883,Z 602.81,A -85,B 0,C 180,E1 23141.568,E2 23141.568} C_VEL
LIN {X 0,Y 112.08,Z 604.039,A -85,B 0,C 180,E1 23149.456,E2 23149.456} C_VEL
LIN {X 0,Y 119.781,Z 623.51,A -85,B 0,C 180,E1 23155.293,E2 23155.293} C_VEL
LIN {X 0,Y 122.862,Z 656.439,A -85,B 0,C 180,E1 23161.56,E2 23161.56} C_VEL
LIN {X 0,Y 132.733,Z 701.582,A -85,B 0,C 180,E1 23173.757,E2 23173.757} C_VEL
LIN {X 0,Y 116.787,Z 750.746,A -85,B 0,C 180,E1 23189.775,E2 23189.775} C_VEL
LIN {X 0,Y 108.98,Z 785.043,A -85,B 0,C 180,E1 23212.002,E2 23212.002} C_VEL
LIN {X 0,Y 112.049,Z 806.203,A -85,B 0,C 180,E1 23237.748,E2 23237.748} C_VEL
LIN {X 0,Y 136.734,Z 817.955,A -85,B 0,C 180,E1 23261.618,E2 23261.618} C_VEL
LIN {X 0,Y 111.278,Z 813.867,A -85,B 0,C 180,E1 23290.136,E2 23290.136} C_VEL
LIN {X 0,Y 110.738,Z 802.705,A -85,B 0,C 180,E1 23312.027,E2 23312.027} C_VEL
LIN {X 0,Y 115.035,Z 776.28,A -85,B 0,C 180,E1 23335.453,E2 23335.453} C_VEL
LIN {X 0,Y 143.725,Z 774.247,A -85,B 0,C 180,E1 23362.435,E2 23362.435} C_VEL
LIN {X 0,Y 117.359,Z 754.279,A -85,B 0,C 180,E1 23383.08,E2 23383.08} C_VEL
LIN {X 0,Y 110.961,Z 722.845,A -85,B 0,C 180,E1 23404.897,E2 23404.897} C_VEL
LIN {X 0,Y 115.142,Z 680.696,A -85,B 0,C 180,E1 23421.878,E2 23421.878} C_VEL
LIN {X 0,Y 115.225,Z 658.559,A -85,B 0,C 180,E1 23427.601,E2 23427.601} C_VEL
LIN {X 0,Y 102.635,Z 602.81,A -85,B 0,C 180,E1 23439.052,E2 23439.052} C_VEL
LIN {X 0,Y 102.153,Z 602.81,A -85,B 0,C 180,E1 23458.594,E2 23458.594} C_VEL
LIN {X 0,Y 104.322,Z 602.81,A -85,B 0,C 180,E1 23477.328,E2 23477.328} C_VEL
LIN {X 0,Y 105.98,Z 602.81,A -85,B 0,C 180,E1 23494.038,E2 23494.038} C_VEL
LIN {X 0,Y 104.437,Z 604.536,A -85,B 0,C 180,E1 23506.2,E2 23506.2} C_VEL
LIN {X 0,Y 122.862,Z 656.439,A -85,B 0,C 180,E1 23521.56,E2 23521.56} C_VEL
LIN {X 0,Y 122.564,Z 688.645,A -85,B 0,C 180,E1 23528.688,E2 23528.688} C_VEL
LIN {X 0,Y 123.314,Z 707.122,A -85,B 0,C 180,E1 23533.934,E2 23533.934} C_VEL
LIN {X 0,Y 107.423,Z 754.506,A -85,B 0,C 180,E1 23551.533,E2 23551.533} C_VEL
LIN {X 0,Y 100.849,Z 787.164,A -85,B 0,C 180,E1 23575.692,E2 23575.692} C_VEL
LIN {X 0,Y 107.933,Z 808.425,A -85,B 0,C 180,E1 23604.954,E2 23604.954} C_VEL
LIN {X 0,Y 127.116,Z 816.943,A -85,B 0,C 180,E1 23621.935,E2 23621.935} C_VEL
LIN {X 0,Y 102.493,Z 808.63,A -85,B 0,C 180,E1 23657.24,E2 23657.24} C_VEL
LIN {X 0,Y 102.948,Z 798.124,A -85,B 0,C 180,E1 23674.295,E2 23674.295} C_VEL
LIN {X 0,Y 107.835,Z 773.071,A -85,B 0,C 180,E1 23696.159,E2 23696.159} C_VEL
LIN {X 0,Y 133.461,Z 772.472,A -85,B 0,C 180,E1 23723.185,E2 23723.185} C_VEL
LIN {X 0,Y 107.945,Z 749.714,A -85,B 0,C 180,E1 23744.711,E2 23744.711} C_VEL
LIN {X 0,Y 103.172,Z 716.015,A -85,B 0,C 180,E1 23767.388,E2 23767.388} C_VEL
LIN {X 0,Y 108.727,Z 670.133,A -85,B 0,C 180,E1 23784.937,E2 23784.937} C_VEL
LIN {X 0,Y 98.505,Z 619.101,A -85,B 0,C 180,E1 23796.249,E2 23796.249} C_VEL
LIN {X 0,Y 94.487,Z 602.81,A -85,B 0,C 180,E1 23800.064,E2 23800.064} C_VEL
LIN {X 0,Y 94.651,Z 602.81,A -85,B 0,C 180,E1 23826.291,E2 23826.291} C_VEL
LIN {X 0,Y 97.64,Z 602.81,A -85,B 0,C 180,E1 23845.471,E2 23845.471} C_VEL
LIN {X 0,Y 96.891,Z 604.679,A -85,B 0,C 180,E1 23862.36,E2 23862.36} C_VEL
LIN {X 0,Y 114.313,Z 653.676,A -85,B 0,C 180,E1 23878.692,E2 23878.692} C_VEL
LIN {X 0,Y 122.564,Z 688.645,A -85,B 0,C 180,E1 23888.688,E2 23888.688} C_VEL
LIN {X 0,Y 114.864,Z 709.269,A -85,B 0,C 180,E1 23893.306,E2 23893.306} C_VEL
LIN {X 0,Y 99.268,Z 754.374,A -85,B 0,C 180,E1 23911.472,E2 23911.472} C_VEL
LIN {X 0,Y 93.042,Z 786.969,A -85,B 0,C 180,E1 23937.671,E2 23937.671} C_VEL
LIN {X 0,Y 103.813,Z 809.352,A -85,B 0,C 180,E1 23970.779,E2 23970.779} C_VEL
LIN {X 0,Y 116.649,Z 815.344,A -85,B 0,C 180,E1 23983.064,E2 23983.064} C_VEL
LIN {X 0,Y 94.954,Z 804.062,A -85,B 0,C 180,E1 24020.88,E2 24020.88} C_VEL
LIN {X 0,Y 95.262,Z 791.902,A -85,B 0,C 180,E1 24038.087,E2 24038.087} C_VEL
LIN {X 0,Y 100.783,Z 769.591,A -85,B 0,C 180,E1 24056.93,E2 24056.93} C_VEL
LIN {X 0,Y 123.055,Z 770.336,A -85,B 0,C 180,E1 24083.025,E2 24083.025} C_VEL
LIN {X 0,Y 98.884,Z 744.299,A -85,B 0,C 180,E1 24106.685,E2 24106.685} C_VEL
LIN {X 0,Y 95.844,Z 707.162,A -85,B 0,C 180,E1 24130.83,E2 24130.83} C_VEL
LIN {X 0,Y 100.32,Z 665.701,A -85,B 0,C 180,E1 24146.339,E2 24146.339} C_VEL
LIN {X 0,Y 88.378,Z 611.3,A -85,B 0,C 180,E1 24158.784,E2 24158.784} C_VEL
LIN {X 0,Y 86.215,Z 602.81,A -85,B 0,C 180,E1 24162.026,E2 24162.026} C_VEL
LIN {X 0,Y 86.327,Z 602.81,A -85,B 0,C 180,E1 24183.842,E2 24183.842} C_VEL
LIN {X 0,Y 89.389,Z 602.81,A -85,B 0,C 180,E1 24205.052,E2 24205.052} C_VEL
LIN {X 0,Y 89.243,Z 604.356,A -85,B 0,C 180,E1 24217.553,E2 24217.553} C_VEL
LIN {X 0,Y 105.524,Z 649.849,A -85,B 0,C 180,E1 24235.084,E2 24235.084} C_VEL
LIN {X 0,Y 116.509,Z 698.712,A -85,B 0,C 180,E1 24250.328,E2 24250.328} C_VEL
LIN {X 0,Y 114.864,Z 709.269,A -85,B 0,C 180,E1 24253.306,E2 24253.306} C_VEL
LIN {X 0,Y 97.592,Z 736.12,A -85,B 0,C 180,E1 24261.838,E2 24261.838} C_VEL
LIN {X 0,Y 85.933,Z 775.626,A -85,B 0,C 180,E1 24288.173,E2 24288.173} C_VEL
LIN {X 0,Y 87.177,Z 797.425,A -85,B 0,C 180,E1 24315.144,E2 24315.144} C_VEL
LIN {X 0,Y 107.105,Z 813.054,A -85,B 0,C 180,E1 24343.005,E2 24343.005} C_VEL
LIN {X 0,Y 87.676,Z 800.152,A -85,B 0,C 180,E1 24382.624,E2 24382.624} C_VEL
LIN {X 0,Y 87.777,Z 784.8,A -85,B 0,C 180,E1 24402.562,E2 24402.562} C_VEL
LIN {X 0,Y 94.194,Z 766.053,A -85,B 0,C 180,E1 24418.985,E2 24418.985} C_VEL
LIN {X 0,Y 112.889,Z 767.56,A -85,B 0,C 180,E1 24442.771,E2 24442.771} C_VEL
LIN {X 0,Y 90.012,Z 738.006,A -85,B 0,C 180,E1 24469.059,E2 24469.059} C_VEL
LIN {X 0,Y 88.844,Z 698.301,A -85,B 0,C 180,E1 24494.205,E2 24494.205} C_VEL
LIN {X 0,Y 91.656,Z 662.937,A -85,B 0,C 180,E1 24507.341,E2 24507.341} C_VEL
LIN {X 0,Y 78.93,Z 606.194,A -85,B 0,C 180,E1 24521.184,E2 24521.184} C_VEL
LIN {X 0,Y 78.093,Z 602.81,A -85,B 0,C 180,E1 24522.84,E2 24522.84} C_VEL
LIN {X 0,Y 79.206,Z 602.81,A -85,B 0,C 180,E1 24553.207,E2 24553.207} C_VEL
LIN {X 0,Y 81.552,Z 604.923,A -85,B 0,C 180,E1 24571.749,E2 24571.749} C_VEL
LIN {X 0,Y 95.387,Z 640.643,A -85,B 0,C 180,E1 24589.074,E2 24589.074} C_VEL
LIN {X 0,Y 107.001,Z 689.767,A -85,B 0,C 180,E1 24605.718,E2 24605.718} C_VEL
LIN {X 0,Y 107.777,Z 707.601,A -85,B 0,C 180,E1 24611.593,E2 24611.593} C_VEL
LIN {X 0,Y 97.592,Z 736.12,A -85,B 0,C 180,E1 24621.838,E2 24621.838} C_VEL
LIN {X 0,Y 81.382,Z 759.501,A -85,B 0,C 180,E1 24635.592,E2 24635.592} C_VEL
LIN {X 0,Y 77.77,Z 788.156,A -85,B 0,C 180,E1 24665.608,E2 24665.608} C_VEL
LIN {X 0,Y 96.48,Z 809.572,A -85,B 0,C 180,E1 24701.327,E2 24701.327} C_VEL
LIN {X 0,Y 92.886,Z 809.116,A -85,B 0,C 180,E1 24707.332,E2 24707.332} C_VEL
LIN {X 0,Y 80.601,Z 794.279,A -85,B 0,C 180,E1 24747.391,E2 24747.391} C_VEL
LIN {X 0,Y 87.891,Z 762.266,A -85,B 0,C 180,E1 24781.287,E2 24781.287} C_VEL
LIN {X 0,Y 102.991,Z 764.037,A -85,B 0,C 180,E1 24802.415,E2 24802.415} C_VEL
LIN {X 0,Y 81.493,Z 732.191,A -85,B 0,C 180,E1 24830.614,E2 24830.614} C_VEL
LIN {X 0,Y 81.584,Z 690.831,A -85,B 0,C 180,E1 24856.848,E2 24856.848} C_VEL
LIN {X 0,Y 83.579,Z 663.078,A -85,B 0,C 180,E1 24867.473,E2 24867.473} C_VEL
LIN {X 0,Y 70.874,Z 606.656,A -85,B 0,C 180,E1 24882.665,E2 24882.665} C_VEL
LIN {X 0,Y 69.906,Z 602.81,A -85,B 0,C 180,E1 24885.761,E2 24885.761} C_VEL
LIN {X 0,Y 72.142,Z 603.65,A -85,B 0,C 180,E1 24921.07,E2 24921.07} C_VEL
LIN {X 0,Y 81.254,Z 620.291,A -85,B 0,C 180,E1 24935.942,E2 24935.942} C_VEL
LIN {X 0,Y 94.111,Z 663.978,A -85,B 0,C 180,E1 24954.384,E2 24954.384} C_VEL
LIN {X 0,Y 100.733,Z 705.954,A -85,B 0,C 180,E1 24969.703,E2 24969.703} C_VEL
LIN {X 0,Y 83.664,Z 751.782,A -85,B 0,C 180,E1 24990.089,E2 24990.089} C_VEL
LIN {X 0,Y 81.382,Z 759.501,A -85,B 0,C 180,E1 24995.592,E2 24995.592} C_VEL
LIN {X 0,Y 69.956,Z 778.792,A -85,B 0,C 180,E1 25016.772,E2 25016.772} C_VEL
LIN {X 0,Y 82.475,Z 803.465,A -85,B 0,C 180,E1 25056.735,E2 25056.735} C_VEL
LIN {X 0,Y 87.39,Z 806.639,A -85,B 0,C 180,E1 25063.914,E2 25063.914} C_VEL
LIN {X 0,Y 73.185,Z 791.002,A -85,B 0,C 180,E1 25107.126,E2 25107.126} C_VEL
LIN {X 0,Y 81.555,Z 758.141,A -85,B 0,C 180,E1 25143.128,E2 25143.128} C_VEL
LIN {X 0,Y 94,Z 760.442,A -85,B 0,C 180,E1 25161.477,E2 25161.477} C_VEL
LIN {X 0,Y 73.16,Z 725.636,A -85,B 0,C 180,E1 25192.542,E2 25192.542} C_VEL
LIN {X 0,Y 74.544,Z 682.364,A -85,B 0,C 180,E1 25219.98,E2 25219.98} C_VEL
LIN {X 0,Y 75.058,Z 661.239,A -85,B 0,C 180,E1 25228.27,E2 25228.27} C_VEL
LIN {X 0,Y 61.605,Z 602.81,A -85,B 0,C 180,E1 25247.764,E2 25247.764} C_VEL
LIN {X 0,Y 70.49,Z 613.563,A -85,B 0,C 180,E1 25283.022,E2 25283.022} C_VEL
LIN {X 0,Y 78.633,Z 632.775,A -85,B 0,C 180,E1 25297.402,E2 25297.402} C_VEL
LIN {X 0,Y 89.362,Z 677.443,A -85,B 0,C 180,E1 25316.704,E2 25316.704} C_VEL
LIN {X 0,Y 92.44,Z 707.701,A -85,B 0,C 180,E1 25328.64,E2 25328.64} C_VEL
LIN {X 0,Y 74.984,Z 753.109,A -85,B 0,C 180,E1 25351.284,E2 25351.284} C_VEL
LIN {X 0,Y 69.956,Z 778.792,A -85,B 0,C 180,E1 25376.772,E2 25376.772} C_VEL
LIN {X 0,Y 66.713,Z 792.731,A -85,B 0,C 180,E1 25404.469,E2 25404.469} C_VEL
LIN {X 0,Y 78.608,Z 802.743,A -85,B 0,C 180,E1 25422.517,E2 25422.517} C_VEL
LIN {X 0,Y 66,Z 789.28,A -85,B 0,C 180,E1 25463.507,E2 25463.507} C_VEL
LIN {X 0,Y 75.768,Z 753.911,A -85,B 0,C 180,E1 25506.034,E2 25506.034} C_VEL
LIN {X 0,Y 84.409,Z 755.506,A -85,B 0,C 180,E1 25520.997,E2 25520.997} C_VEL
LIN {X 0,Y 65.408,Z 720.207,A -85,B 0,C 180,E1 25553.328,E2 25553.328} C_VEL
LIN {X 0,Y 67.532,Z 675.457,A -85,B 0,C 180,E1 25582.487,E2 25582.487} C_VEL
LIN {X 0,Y 64.355,Z 648.547,A -85,B 0,C 180,E1 25592.989,E2 25592.989} C_VEL
LIN {X 0,Y 57.655,Z 615.488,A -85,B 0,C 180,E1 25605.867,E2 25605.867} C_VEL
LIN {X 0,Y 59.116,Z 611.481,A -85,B 0,C 180,E1 25612.95,E2 25612.95} C_VEL
LIN {X 0,Y 67.767,Z 621.567,A -85,B 0,C 180,E1 25642.74,E2 25642.74} C_VEL
LIN {X 0,Y 76.249,Z 648.993,A -85,B 0,C 180,E1 25660.658,E2 25660.658} C_VEL
LIN {X 0,Y 84.61,Z 695.229,A -85,B 0,C 180,E1 25681.564,E2 25681.564} C_VEL
LIN {X 0,Y 83.794,Z 710.33,A -85,B 0,C 180,E1 25687.762,E2 25687.762} C_VEL
LIN {X 0,Y 65.836,Z 756.112,A -85,B 0,C 180,E1 25714.406,E2 25714.406} C_VEL
LIN {X 0,Y 62.876,Z 783.735,A -85,B 0,C 180,E1 25748.674,E2 25748.674} C_VEL
LIN {X 0,Y 66.713,Z 792.731,A -85,B 0,C 180,E1 25764.469,E2 25764.469} C_VEL
LIN {X 0,Y 70.54,Z 798.427,A -85,B 0,C 180,E1 25779.312,E2 25779.312} C_VEL
LIN {X 0,Y 69.321,Z 798.393,A -85,B 0,C 180,E1 25784.073,E2 25784.073} C_VEL
LIN {X 0,Y 58.495,Z 783.751,A -85,B 0,C 180,E1 25826.403,E2 25826.403} C_VEL
LIN {X 0,Y 68.115,Z 750.661,A -85,B 0,C 180,E1 25866.451,E2 25866.451} C_VEL
LIN {X 0,Y 75.832,Z 750.754,A -85,B 0,C 180,E1 25879.417,E2 25879.417} C_VEL
LIN {X 0,Y 57.763,Z 714.171,A -85,B 0,C 180,E1 25914.334,E2 25914.334} C_VEL
LIN {X 0,Y 60.288,Z 670.041,A -85,B 0,C 180,E1 25944.499,E2 25944.499} C_VEL
LIN {X 0,Y 53.211,Z 632.219,A -85,B 0,C 180,E1 25962.189,E2 25962.189} C_VEL
LIN {X 0,Y 56.962,Z 620.023,A -85,B 0,C 180,E1 25974.395,E2 25974.395} C_VEL
LIN {X 0,Y 64.41,Z 628.609,A -85,B 0,C 180,E1 26001.137,E2 26001.137} C_VEL
LIN {X 0,Y 72.27,Z 662.489,A -85,B 0,C 180,E1 26022.789,E2 26022.789} C_VEL
LIN {X 0,Y 77.965,Z 705.947,A -85,B 0,C 180,E1 26044.188,E2 26044.188} C_VEL
LIN {X 0,Y 58.924,Z 751.59,A -85,B 0,C 180,E1 26071.14,E2 26071.14} C_VEL
LIN {X 0,Y 55.479,Z 780.722,A -85,B 0,C 180,E1 26109.856,E2 26109.856} C_VEL
LIN {X 0,Y 69.321,Z 798.393,A -85,B 0,C 180,E1 26144.073,E2 26144.073} C_VEL
LIN {X 0,Y 52.058,Z 785.62,A -85,B 0,C 180,E1 26171.424,E2 26171.424} C_VEL
LIN {X 0,Y 50.105,Z 773.438,A -85,B 0,C 180,E1 26196.663,E2 26196.663} C_VEL
LIN {X 0,Y 64.605,Z 744.603,A -85,B 0,C 180,E1 26231.585,E2 26231.585} C_VEL
LIN {X 0,Y 66.373,Z 744.111,A -85,B 0,C 180,E1 26238.89,E2 26238.89} C_VEL
LIN {X 0,Y 49.744,Z 705.05,A -85,B 0,C 180,E1 26277.801,E2 26277.801} C_VEL
LIN {X 0,Y 51.575,Z 665.37,A -85,B 0,C 180,E1 26306.175,E2 26306.175} C_VEL
LIN {X 0,Y 48.668,Z 649.67,A -85,B 0,C 180,E1 26316.794,E2 26316.794} C_VEL
LIN {X 0,Y 55.101,Z 629.04,A -85,B 0,C 180,E1 26338.177,E2 26338.177} C_VEL
LIN {X 0,Y 60.966,Z 635.875,A -85,B 0,C 180,E1 26359.268,E2 26359.268} C_VEL
LIN {X 0,Y 66.769,Z 671.924,A -85,B 0,C 180,E1 26383.026,E2 26383.026} C_VEL
LIN {X 0,Y 69.947,Z 707.157,A -85,B 0,C 180,E1 26402.23,E2 26402.23} C_VEL
LIN {X 0,Y 50.019,Z 753.6,A -85,B 0,C 180,E1 26434.449,E2 26434.449} C_VEL
LIN {X 0,Y 49.169,Z 780.439,A -85,B 0,C 180,E1 26477.409,E2 26477.409} C_VEL
LIN {X 0,Y 60.443,Z 793.55,A -85,B 0,C 180,E1 26505.059,E2 26505.059} C_VEL
LIN {X 0,Y 52.058,Z 785.62,A -85,B 0,C 180,E1 26531.424,E2 26531.424} C_VEL
LIN {X 0,Y 46.973,Z 776.435,A -85,B 0,C 180,E1 26547.611,E2 26547.611} C_VEL
LIN {X 0,Y 43.03,Z 764.457,A -85,B 0,C 180,E1 26565.282,E2 26565.282} C_VEL
LIN {X 0,Y 59.124,Z 738.985,A -85,B 0,C 180,E1 26595.849,E2 26595.849} C_VEL
LIN {X 0,Y 42.252,Z 698.575,A -85,B 0,C 180,E1 26638.698,E2 26638.698} C_VEL
LIN {X 0,Y 43.931,Z 667.232,A -85,B 0,C 180,E1 26667.934,E2 26667.934} C_VEL
LIN {X 0,Y 53.577,Z 637.744,A -85,B 0,C 180,E1 26702.475,E2 26702.475} C_VEL
LIN {X 0,Y 57.372,Z 643.516,A -85,B 0,C 180,E1 26717.325,E2 26717.325} C_VEL
LIN {X 0,Y 61.099,Z 682.395,A -85,B 0,C 180,E1 26744.26,E2 26744.26} C_VEL
LIN {X 0,Y 61.508,Z 709.361,A -85,B 0,C 180,E1 26760.311,E2 26760.311} C_VEL
LIN {X 0,Y 41.388,Z 754.82,A -85,B 0,C 180,E1 26798.35,E2 26798.35} C_VEL
LIN {X 0,Y 44.288,Z 780.511,A -85,B 0,C 180,E1 26848.125,E2 26848.125} C_VEL
LIN {X 0,Y 51.544,Z 788.041,A -85,B 0,C 180,E1 26866.634,E2 26866.634} C_VEL
LIN {X 0,Y 43.844,Z 775.525,A -85,B 0,C 180,E1 26905.199,E2 26905.199} C_VEL
LIN {X 0,Y 43.03,Z 764.457,A -85,B 0,C 180,E1 26925.282,E2 26925.282} C_VEL
LIN {X 0,Y 42.21,Z 747.12,A -85,B 0,C 180,E1 26947.697,E2 26947.697} C_VEL
LIN {X 0,Y 48.774,Z 737.937,A -85,B 0,C 180,E1 26956.883,E2 26956.883} C_VEL
LIN {X 0,Y 36.566,Z 689.961,A -85,B 0,C 180,E1 27016.332,E2 27016.332} C_VEL
LIN {X 0,Y 40.495,Z 672.797,A -85,B 0,C 180,E1 27034.181,E2 27034.181} C_VEL
LIN {X 0,Y 51.011,Z 646.9,A -85,B 0,C 180,E1 27063.345,E2 27063.345} C_VEL
LIN {X 0,Y 53.368,Z 648.878,A -85,B 0,C 180,E1 27072.711,E2 27072.711} C_VEL
LIN {X 0,Y 54.742,Z 687.848,A -85,B 0,C 180,E1 27102.468,E2 27102.468} C_VEL
LIN {X 0,Y 54.109,Z 709.369,A -85,B 0,C 180,E1 27116.884,E2 27116.884} C_VEL
LIN {X 0,Y 33.243,Z 754.164,A -85,B 0,C 180,E1 27161.166,E2 27161.166} C_VEL
LIN {X 0,Y 38.942,Z 778.08,A -85,B 0,C 180,E1 27215.79,E2 27215.79} C_VEL
LIN {X 0,Y 43.474,Z 782.318,A -85,B 0,C 180,E1 27225.174,E2 27225.174} C_VEL
LIN {X 0,Y 36.969,Z 772.295,A -85,B 0,C 180,E1 27261.34,E2 27261.34} C_VEL
LIN {X 0,Y 42.21,Z 747.12,A -85,B 0,C 180,E1 27307.697,E2 27307.697} C_VEL
LIN {X 0,Y 40.691,Z 738.595,A -85,B 0,C 180,E1 27317.15,E2 27317.15} C_VEL
LIN {X 0,Y 33.976,Z 729.632,A -85,B 0,C 180,E1 27329.348,E2 27329.348} C_VEL
LIN {X 0,Y 37.983,Z 676.789,A -85,B 0,C 180,E1 27404.212,E2 27404.212} C_VEL
LIN {X 0,Y 49.541,Z 656.124,A -85,B 0,C 180,E1 27429.316,E2 27429.316} C_VEL
LIN {X 0,Y 48.251,Z 696.647,A -85,B 0,C 180,E1 27463.032,E2 27463.032} C_VEL
LIN {X 0,Y 45.926,Z 711.189,A -85,B 0,C 180,E1 27473.42,E2 27473.42} C_VEL
LIN {X 0,Y 25.06,Z 755.515,A -85,B 0,C 180,E1 27531.321,E2 27531.321} C_VEL
LIN {X 0,Y 33.404,Z 774.344,A -85,B 0,C 180,E1 27582.983,E2 27582.983} C_VEL
LIN {X 0,Y 35.162,Z 775.959,A -85,B 0,C 180,E1 27589.925,E2 27589.925} C_VEL
LIN {X 0,Y 29.762,Z 767.547,A -85,B 0,C 180,E1 27619.221,E2 27619.221} C_VEL
LIN {X 0,Y 38.608,Z 736.991,A -85,B 0,C 180,E1 27679.2,E2 27679.2} C_VEL
LIN {X 0,Y 33.976,Z 729.632,A -85,B 0,C 180,E1 27689.348,E2 27689.348} C_VEL
LIN {X 0,Y 24.628,Z 707.438,A -85,B 0,C 180,E1 27742.816,E2 27742.816} C_VEL
LIN {X 0,Y 37.312,Z 679.494,A -85,B 0,C 180,E1 27776.753,E2 27776.753} C_VEL
LIN {X 0,Y 44.879,Z 668.328,A -85,B 0,C 180,E1 27790.102,E2 27790.102} C_VEL
LIN {X 0,Y 41.108,Z 707.309,A -85,B 0,C 180,E1 27825.771,E2 27825.771} C_VEL
LIN {X 0,Y 17.698,Z 752.261,A -85,B 0,C 180,E1 27893.886,E2 27893.886} C_VEL
LIN {X 0,Y 27.082,Z 769.049,A -85,B 0,C 180,E1 27949.394,E2 27949.394} C_VEL
LIN {X 0,Y 23.48,Z 763.909,A -85,B 0,C 180,E1 27971.467,E2 27971.467} C_VEL
LIN {X 0,Y 29.212,Z 736.855,A -85,B 0,C 180,E1 28041.283,E2 28041.283} C_VEL
LIN {X 0,Y 24.628,Z 707.438,A -85,B 0,C 180,E1 28102.816,E2 28102.816} C_VEL
LIN {X 0,Y 31.453,Z 692.234,A -85,B 0,C 180,E1 28138.964,E2 28138.964} C_VEL
LIN {X 0,Y 39.014,Z 682.243,A -85,B 0,C 180,E1 28151.862,E2 28151.862} C_VEL
LIN {X 0,Y 32.983,Z 710.061,A -85,B 0,C 180,E1 28179.131,E2 28179.131} C_VEL
LIN {X 0,Y 12.385,Z 753.826,A -85,B 0,C 180,E1 28287.416,E2 28287.416} C_VEL
LIN {X 0,Y 18.44,Z 760.74,A -85,B 0,C 180,E1 28316.731,E2 28316.731} C_VEL
LIN {X 0,Y 19.952,Z 736.932,A -85,B 0,C 180,E1 28404.254,E2 28404.254} C_VEL
LIN {X 0,Y 31.453,Z 692.234,A -85,B 0,C 180,E1 28498.964,E2 28498.964} C_VEL
LIN {X 0,Y 31.478,Z 697.103,A -85,B 0,C 180,E1 28513.731,E2 28513.731} C_VEL
LIN {X 0,Y 30.622,Z 700.818,A -85,B 0,C 180,E1 28518.759,E2 28518.759} C_VEL
LIN {X 0,Y 25.629,Z 712.432,A -85,B 0,C 180,E1 28528.356,E2 28528.356} C_VEL
LIN {X 0,Y 7.224,Z 748.867,A -85,B 0,C 180,E1 28677.444,E2 28677.444} C_VEL
LIN {X 0,Y 10.789,Z 736.782,A -85,B 0,C 180,E1 28772.262,E2 28772.262} C_VEL
LIN {X 0,Y 31.765,Z 696.697,A -85,B 0,C 180,E1 28873.992,E2 28873.992} C_VEL
LIN {X 0,Y 30.622,Z 700.818,A -85,B 0,C 180,E1 28878.759,E2 28878.759} C_VEL
LIN {X 0,Y 30.477,Z 701.957,A -85,B 0,C 180,E1 28879.368,E2 28879.368} C_VEL
LIN {X 0,Y 30.477,Z 855,A -85,B 0,C 180,E1 28879.368,E2 28879.368} C_VEL
LIN {X 0,Y 30.477,Z 855,A -85,B 0,C 180,E1 28879.368,E2 28879.368}

